LIN {X 0,Y 511.313,Z 919.131,A -85,B 0,C 180,E1 -11823.667,E2 -11823.667} C_VEL
LIN {X 0,Y 515.033,Z 901.309,A -85,B 0,C 180,E1 -11825.28,E2 -11825.28} C_VEL
LIN {X 0,Y 519.279,Z 879.68,A -85,B 0,C 180,E1 -11826.956,E2 -11826.956} C_VEL
LIN {X 0,Y 522.584,Z 861.401,A -85,B 0,C 180,E1 -11828.171,E2 -11828.171} C_VEL
LIN {X 0,Y 526.187,Z 839.915,A -85,B 0,C 180,E1 -11829.397,E2 -11829.397} C_VEL
LIN {X 0,Y 529.318,Z 818.14,A -85,B 0,C 180,E1 -11830.423,E2 -11830.423} C_VEL
LIN {X 0,Y 532.01,Z 796.933,A -85,B 0,C 180,E1 -11831.255,E2 -11831.255} C_VEL
LIN {X 0,Y 534.495,Z 772.49,A -85,B 0,C 180,E1 -11832.005,E2 -11832.005} C_VEL
LIN {X 0,Y 536.169,Z 751.43,A -85,B 0,C 180,E1 -11832.497,E2 -11832.497} C_VEL
LIN {X 0,Y 537.704,Z 719.028,A -85,B 0,C 180,E1 -11833.031,E2 -11833.031} C_VEL
LIN {X 0,Y 546.817,Z 464.332,A -85,B 0,C 180,E1 -11836.745,E2 -11836.745} C_VEL
LIN {X 0,Y 547.523,Z 441.329,A -85,B 0,C 180,E1 -11837.1,E2 -11837.1} C_VEL
LIN {X 0,Y 534.412,Z 419.937,A -85,B 0,C 180,E1 -11839.073,E2 -11839.073} C_VEL
LIN {X 0,Y 522.198,Z 402.674,A -85,B 0,C 180,E1 -11841.023,E2 -11841.023} C_VEL
LIN {X 0,Y 514.394,Z 392.307,A -85,B 0,C 180,E1 -11842.349,E2 -11842.349} C_VEL
LIN {X 0,Y 507.087,Z 382.771,A -85,B 0,C 180,E1 -11843.663,E2 -11843.663} C_VEL
LIN {X 0,Y 502.805,Z 377.333,A -85,B 0,C 180,E1 -11844.467,E2 -11844.467} C_VEL
LIN {X 0,Y 499.561,Z 373.172,A -85,B 0,C 180,E1 -11845.097,E2 -11845.097} C_VEL
LIN {X 0,Y 498.35,Z 371.8,A -85,B 0,C 180,E1 -11845.332,E2 -11845.332} C_VEL
LIN {X 0,Y 495.465,Z 368.374,A -85,B 0,C 180,E1 -11845.908,E2 -11845.908} C_VEL
LIN {X 0,Y 494.414,Z 366.395,A -85,B 0,C 180,E1 -11846.14,E2 -11846.14} C_VEL
LIN {X 0,Y 491.49,Z 364.03,A -85,B 0,C 180,E1 -11846.716,E2 -11846.716} C_VEL
LIN {X 0,Y 490.096,Z 361.064,A -85,B 0,C 180,E1 -11847.046,E2 -11847.046} C_VEL
LIN {X 0,Y 489.943,Z 360.201,A -85,B 0,C 180,E1 -11847.121,E2 -11847.121} C_VEL
LIN {X 0,Y 489.937,Z 360.204,A -85,B 0,C 180,E1 -11850.672,E2 -11850.672} C_VEL
LIN {X 0,Y 489.975,Z 360.197,A -85,B 0,C 180,E1 -11854.106,E2 -11854.106} C_VEL
LIN {X 0,Y 489.965,Z 360.19,A -85,B 0,C 180,E1 -11857.586,E2 -11857.586} C_VEL
LIN {X 0,Y 489.933,Z 360.182,A -85,B 0,C 180,E1 -11861.065,E2 -11861.065} C_VEL
LIN {X 0,Y 489.943,Z 360.174,A -85,B 0,C 180,E1 -11864.615,E2 -11864.615} C_VEL
LIN {X 0,Y 489.979,Z 360.18,A -85,B 0,C 180,E1 -11867.986,E2 -11867.986} C_VEL
LIN {X 0,Y 489.937,Z 360.202,A -85,B 0,C 180,E1 -11871.432,E2 -11871.432} C_VEL
LIN {X 0,Y 489.932,Z 360.192,A -85,B 0,C 180,E1 -11875.083,E2 -11875.083} C_VEL
LIN {X 0,Y 489.976,Z 360.169,A -85,B 0,C 180,E1 -11878.48,E2 -11878.48} C_VEL
LIN {X 0,Y 489.95,Z 360.185,A -85,B 0,C 180,E1 -11881.871,E2 -11881.871} C_VEL
LIN {X 0,Y 489.931,Z 360.202,A -85,B 0,C 180,E1 -11885.387,E2 -11885.387} C_VEL
LIN {X 0,Y 489.963,Z 360.181,A -85,B 0,C 180,E1 -11888.804,E2 -11888.804} C_VEL
LIN {X 0,Y 489.967,Z 360.172,A -85,B 0,C 180,E1 -11892.253,E2 -11892.253} C_VEL
LIN {X 0,Y 489.93,Z 360.186,A -85,B 0,C 180,E1 -11895.628,E2 -11895.628} C_VEL
LIN {X 0,Y 489.946,Z 360.196,A -85,B 0,C 180,E1 -11899.182,E2 -11899.182} C_VEL
LIN {X 0,Y 490,Z 360.194,A -85,B 0,C 180,E1 -11902.686,E2 -11902.686} C_VEL
LIN {X 0,Y 489.945,Z 360.2,A -85,B 0,C 180,E1 -11906.156,E2 -11906.156} C_VEL
LIN {X 0,Y 489.937,Z 360.204,A -85,B 0,C 180,E1 -11909.611,E2 -11909.611} C_VEL
LIN {X 0,Y 489.959,Z 360.296,A -85,B 0,C 180,E1 -11911.399,E2 -11911.399} C_VEL
LIN {X 0,Y 491.112,Z 363.479,A -85,B 0,C 180,E1 -11912.117,E2 -11912.117} C_VEL
LIN {X 0,Y 492.216,Z 365.12,A -85,B 0,C 180,E1 -11912.57,E2 -11912.57} C_VEL
LIN {X 0,Y 494.473,Z 369.884,A -85,B 0,C 180,E1 -11913.629,E2 -11913.629} C_VEL
LIN {X 0,Y 497.873,Z 374.385,A -85,B 0,C 180,E1 -11914.322,E2 -11914.322} C_VEL
LIN {X 0,Y 506.25,Z 385.924,A -85,B 0,C 180,E1 -11915.951,E2 -11915.951} C_VEL
LIN {X 0,Y 515.686,Z 399.295,A -85,B 0,C 180,E1 -11917.663,E2 -11917.663} C_VEL
LIN {X 0,Y 526.361,Z 415.198,A -85,B 0,C 180,E1 -11919.469,E2 -11919.469} C_VEL
LIN {X 0,Y 538.606,Z 435.059,A -85,B 0,C 180,E1 -11921.409,E2 -11921.409} C_VEL
LIN {X 0,Y 547.534,Z 450.875,A -85,B 0,C 180,E1 -11922.751,E2 -11922.751} C_VEL
LIN {X 0,Y 538.539,Z 702.351,A -85,B 0,C 180,E1 -11926.422,E2 -11926.422} C_VEL
LIN {X 0,Y 536.196,Z 765.178,A -85,B 0,C 180,E1 -11927.36,E2 -11927.36} C_VEL
LIN {X 0,Y 534.217,Z 790.289,A -85,B 0,C 180,E1 -11927.896,E2 -11927.896} C_VEL
LIN {X 0,Y 532.012,Z 811.704,A -85,B 0,C 180,E1 -11928.504,E2 -11928.504} C_VEL
LIN {X 0,Y 528.819,Z 836.909,A -85,B 0,C 180,E1 -11929.426,E2 -11929.426} C_VEL
LIN {X 0,Y 525.791,Z 857.705,A -85,B 0,C 180,E1 -11930.371,E2 -11930.371} C_VEL
LIN {X 0,Y 521.793,Z 881.818,A -85,B 0,C 180,E1 -11931.69,E2 -11931.69} C_VEL
LIN {X 0,Y 518.363,Z 900.79,A -85,B 0,C 180,E1 -11932.927,E2 -11932.927} C_VEL
LIN {X 0,Y 514.303,Z 921.939,A -85,B 0,C 180,E1 -11934.526,E2 -11934.526} C_VEL
LIN {X 0,Y 510.427,Z 940.778,A -85,B 0,C 180,E1 -11936.197,E2 -11936.197} C_VEL
LIN {X 0,Y 506.569,Z 959.339,A -85,B 0,C 180,E1 -11938.077,E2 -11938.077} C_VEL
LIN {X 0,Y 502.777,Z 977.115,A -85,B 0,C 180,E1 -11940.186,E2 -11940.186} C_VEL
LIN {X 0,Y 499.343,Z 993.821,A -85,B 0,C 180,E1 -11942.448,E2 -11942.448} C_VEL
LIN {X 0,Y 496.299,Z 1008.916,A -85,B 0,C 180,E1 -11944.843,E2 -11944.843} C_VEL
LIN {X 0,Y 493.733,Z 1022.841,A -85,B 0,C 180,E1 -11947.37,E2 -11947.37} C_VEL
LIN {X 0,Y 491.7,Z 1034.931,A -85,B 0,C 180,E1 -11949.968,E2 -11949.968} C_VEL
LIN {X 0,Y 490.163,Z 1045.803,A -85,B 0,C 180,E1 -11952.673,E2 -11952.673} C_VEL
LIN {X 0,Y 489.084,Z 1054.892,A -85,B 0,C 180,E1 -11955.436,E2 -11955.436} C_VEL
LIN {X 0,Y 488.449,Z 1062.177,A -85,B 0,C 180,E1 -11958.099,E2 -11958.099} C_VEL
LIN {X 0,Y 488.077,Z 1068.149,A -85,B 0,C 180,E1 -11960.924,E2 -11960.924} C_VEL
LIN {X 0,Y 487.956,Z 1071.916,A -85,B 0,C 180,E1 -11963.292,E2 -11963.292} C_VEL
LIN {X 0,Y 487.923,Z 1074.916,A -85,B 0,C 180,E1 -11966.005,E2 -11966.005} C_VEL
LIN {X 0,Y 487.926,Z 1076.286,A -85,B 0,C 180,E1 -11968.708,E2 -11968.708} C_VEL
LIN {X 0,Y 487.932,Z 1076.332,A -85,B 0,C 180,E1 -11971.057,E2 -11971.057} C_VEL
LIN {X 0,Y 487.925,Z 1075.157,A -85,B 0,C 180,E1 -11973.642,E2 -11973.642} C_VEL
LIN {X 0,Y 487.952,Z 1072.239,A -85,B 0,C 180,E1 -11976.471,E2 -11976.471} C_VEL
LIN {X 0,Y 488.061,Z 1068.568,A -85,B 0,C 180,E1 -11978.839,E2 -11978.839} C_VEL
LIN {X 0,Y 488.368,Z 1063.239,A -85,B 0,C 180,E1 -11981.455,E2 -11981.455} C_VEL
LIN {X 0,Y 488.988,Z 1055.838,A -85,B 0,C 180,E1 -11984.246,E2 -11984.246} C_VEL
LIN {X 0,Y 489.879,Z 1047.867,A -85,B 0,C 180,E1 -11986.726,E2 -11986.726} C_VEL
LIN {X 0,Y 491.42,Z 1036.727,A -85,B 0,C 180,E1 -11989.617,E2 -11989.617} C_VEL
LIN {X 0,Y 493.107,Z 1026.321,A -85,B 0,C 180,E1 -11991.907,E2 -11991.907} C_VEL
LIN {X 0,Y 495.582,Z 1012.759,A -85,B 0,C 180,E1 -11994.502,E2 -11994.502} C_VEL
LIN {X 0,Y 498.352,Z 998.474,A -85,B 0,C 180,E1 -11996.836,E2 -11996.836} C_VEL
LIN {X 0,Y 501.637,Z 982.689,A -85,B 0,C 180,E1 -11999.101,E2 -11999.101} C_VEL
LIN {X 0,Y 505.249,Z 965.34,A -85,B 0,C 180,E1 -12001.231,E2 -12001.231} C_VEL
LIN {X 0,Y 509.17,Z 946.864,A -85,B 0,C 180,E1 -12003.22,E2 -12003.22} C_VEL
LIN {X 0,Y 513.17,Z 927.247,A -85,B 0,C 180,E1 -12005.017,E2 -12005.017} C_VEL
LIN {X 0,Y 517.179,Z 907.204,A -85,B 0,C 180,E1 -12006.615,E2 -12006.615} C_VEL
LIN {X 0,Y 520.987,Z 886.248,A -85,B 0,C 180,E1 -12008.03,E2 -12008.03} C_VEL
LIN {X 0,Y 524.287,Z 867.033,A -85,B 0,C 180,E1 -12009.143,E2 -12009.143} C_VEL
LIN {X 0,Y 527.961,Z 842.844,A -85,B 0,C 180,E1 -12010.317,E2 -12010.317} C_VEL
LIN {X 0,Y 530.724,Z 822.066,A -85,B 0,C 180,E1 -12011.139,E2 -12011.139} C_VEL
LIN {X 0,Y 533.484,Z 797.595,A -85,B 0,C 180,E1 -12011.913,E2 -12011.913} C_VEL
LIN {X 0,Y 535.471,Z 774.643,A -85,B 0,C 180,E1 -12012.452,E2 -12012.452} C_VEL
LIN {X 0,Y 536.913,Z 748.928,A -85,B 0,C 180,E1 -12012.896,E2 -12012.896} C_VEL
LIN {X 0,Y 545.727,Z 498.186,A -85,B 0,C 180,E1 -12016.55,E2 -12016.55} C_VEL
LIN {X 0,Y 547.401,Z 450.448,A -85,B 0,C 180,E1 -12017.259,E2 -12017.259} C_VEL
LIN {X 0,Y 535.227,Z 429.465,A -85,B 0,C 180,E1 -12019.096,E2 -12019.096} C_VEL
LIN {X 0,Y 523.091,Z 410.309,A -85,B 0,C 180,E1 -12021.049,E2 -12021.049} C_VEL
LIN {X 0,Y 511.933,Z 393.825,A -85,B 0,C 180,E1 -12022.982,E2 -12022.982} C_VEL
LIN {X 0,Y 503.577,Z 382.206,A -85,B 0,C 180,E1 -12024.529,E2 -12024.529} C_VEL
LIN {X 0,Y 496.871,Z 373.305,A -85,B 0,C 180,E1 -12025.843,E2 -12025.843} C_VEL
LIN {X 0,Y 494.047,Z 368.955,A -85,B 0,C 180,E1 -12026.495,E2 -12026.495} C_VEL
LIN {X 0,Y 492.345,Z 365.591,A -85,B 0,C 180,E1 -12027.302,E2 -12027.302} C_VEL
LIN {X 0,Y 490.139,Z 361.244,A -85,B 0,C 180,E1 -12028.38,E2 -12028.38} C_VEL
LIN {X 0,Y 489.946,Z 360.176,A -85,B 0,C 180,E1 -12028.64,E2 -12028.64} C_VEL
LIN {X 0,Y 489.935,Z 360.177,A -85,B 0,C 180,E1 -12032.137,E2 -12032.137} C_VEL
LIN {X 0,Y 489.961,Z 360.177,A -85,B 0,C 180,E1 -12035.655,E2 -12035.655} C_VEL
LIN {X 0,Y 489.96,Z 360.184,A -85,B 0,C 180,E1 -12038.95,E2 -12038.95} C_VEL
LIN {X 0,Y 489.935,Z 360.2,A -85,B 0,C 180,E1 -12042.419,E2 -12042.419} C_VEL
LIN {X 0,Y 489.954,Z 360.203,A -85,B 0,C 180,E1 -12045.945,E2 -12045.945} C_VEL
LIN {X 0,Y 489.983,Z 360.182,A -85,B 0,C 180,E1 -12049.417,E2 -12049.417} C_VEL
LIN {X 0,Y 489.935,Z 360.172,A -85,B 0,C 180,E1 -12052.849,E2 -12052.849} C_VEL
LIN {X 0,Y 489.939,Z 360.185,A -85,B 0,C 180,E1 -12056.373,E2 -12056.373} C_VEL
LIN {X 0,Y 489.986,Z 360.198,A -85,B 0,C 180,E1 -12059.883,E2 -12059.883} C_VEL
LIN {X 0,Y 489.964,Z 360.186,A -85,B 0,C 180,E1 -12063.393,E2 -12063.393} C_VEL
LIN {X 0,Y 489.931,Z 360.174,A -85,B 0,C 180,E1 -12066.798,E2 -12066.798} C_VEL
LIN {X 0,Y 489.965,Z 360.183,A -85,B 0,C 180,E1 -12070.227,E2 -12070.227} C_VEL
LIN {X 0,Y 489.99,Z 360.198,A -85,B 0,C 180,E1 -12073.813,E2 -12073.813} C_VEL
LIN {X 0,Y 489.941,Z 360.194,A -85,B 0,C 180,E1 -12077.233,E2 -12077.233} C_VEL
LIN {X 0,Y 489.943,Z 360.182,A -85,B 0,C 180,E1 -12080.821,E2 -12080.821} C_VEL
LIN {X 0,Y 489.986,Z 360.174,A -85,B 0,C 180,E1 -12084.216,E2 -12084.216} C_VEL
LIN {X 0,Y 489.96,Z 360.178,A -85,B 0,C 180,E1 -12087.729,E2 -12087.729} C_VEL
LIN {X 0,Y 489.937,Z 360.181,A -85,B 0,C 180,E1 -12091.224,E2 -12091.224} C_VEL
LIN {X 0,Y 489.96,Z 360.317,A -85,B 0,C 180,E1 -12093.034,E2 -12093.034} C_VEL
LIN {X 0,Y 490.954,Z 363.217,A -85,B 0,C 180,E1 -12093.29,E2 -12093.29} C_VEL
LIN {X 0,Y 493.433,Z 365.836,A -85,B 0,C 180,E1 -12093.797,E2 -12093.797} C_VEL
LIN {X 0,Y 494.715,Z 366.871,A -85,B 0,C 180,E1 -12094.046,E2 -12094.046} C_VEL
LIN {X 0,Y 497.133,Z 370.66,A -85,B 0,C 180,E1 -12094.555,E2 -12094.555} C_VEL
LIN {X 0,Y 499.453,Z 372.962,A -85,B 0,C 180,E1 -12094.999,E2 -12094.999} C_VEL
LIN {X 0,Y 502.626,Z 377.161,A -85,B 0,C 180,E1 -12095.618,E2 -12095.618} C_VEL
LIN {X 0,Y 504.307,Z 379.254,A -85,B 0,C 180,E1 -12095.936,E2 -12095.936} C_VEL
LIN {X 0,Y 509.417,Z 385.807,A -85,B 0,C 180,E1 -12096.879,E2 -12096.879} C_VEL
LIN {X 0,Y 519.764,Z 399.344,A -85,B 0,C 180,E1 -12098.681,E2 -12098.681} C_VEL
LIN {X 0,Y 532.978,Z 417.831,A -85,B 0,C 180,E1 -12100.811,E2 -12100.811} C_VEL
LIN {X 0,Y 544.745,Z 436.73,A -85,B 0,C 180,E1 -12102.598,E2 -12102.598} C_VEL
LIN {X 0,Y 547.588,Z 441.89,A -85,B 0,C 180,E1 -12103.021,E2 -12103.021} C_VEL
LIN {X 0,Y 538.598,Z 691.495,A -85,B 0,C 180,E1 -12106.663,E2 -12106.663} C_VEL
LIN {X 0,Y 536.531,Z 745.384,A -85,B 0,C 180,E1 -12107.475,E2 -12107.475} C_VEL
LIN {X 0,Y 534.688,Z 769.631,A -85,B 0,C 180,E1 -12108.014,E2 -12108.014} C_VEL
LIN {X 0,Y 532.499,Z 791.967,A -85,B 0,C 180,E1 -12108.669,E2 -12108.669} C_VEL
LIN {X 0,Y 529.612,Z 815.624,A -85,B 0,C 180,E1 -12109.563,E2 -12109.563} C_VEL
LIN {X 0,Y 526.696,Z 836.1,A -85,B 0,C 180,E1 -12110.508,E2 -12110.508} C_VEL
LIN {X 0,Y 522.882,Z 859.553,A -85,B 0,C 180,E1 -12111.808,E2 -12111.808} C_VEL
LIN {X 0,Y 519.541,Z 878.086,A -85,B 0,C 180,E1 -12113.028,E2 -12113.028} C_VEL
LIN {X 0,Y 515.648,Z 898.366,A -85,B 0,C 180,E1 -12114.564,E2 -12114.564} C_VEL
LIN {X 0,Y 511.606,Z 917.639,A -85,B 0,C 180,E1 -12116.286,E2 -12116.286} C_VEL
LIN {X 0,Y 507.757,Z 935.822,A -85,B 0,C 180,E1 -12118.146,E2 -12118.146} C_VEL
LIN {X 0,Y 506.748,Z 940.366,A -85,B 0,C 180,E1 -12118.669,E2 -12118.669} C_VEL
LIN {X 0,Y 504.678,Z 945.91,A -85,B 0,C 180,E1 -12119.252,E2 -12119.252} C_VEL
LIN {X 0,Y 495.934,Z 960.386,A -85,B 0,C 180,E1 -12120.722,E2 -12120.722} C_VEL
LIN {X 0,Y 494.284,Z 964.589,A -85,B 0,C 180,E1 -12121.277,E2 -12121.277} C_VEL
LIN {X 0,Y 490.862,Z 979.995,A -85,B 0,C 180,E1 -12123.636,E2 -12123.636} C_VEL
LIN {X 0,Y 487.931,Z 993.479,A -85,B 0,C 180,E1 -12126.062,E2 -12126.062} C_VEL
LIN {X 0,Y 485.559,Z 1005.29,A -85,B 0,C 180,E1 -12128.497,E2 -12128.497} C_VEL
LIN {X 0,Y 483.479,Z 1016.797,A -85,B 0,C 180,E1 -12131.303,E2 -12131.303} C_VEL
LIN {X 0,Y 482.143,Z 1025.397,A -85,B 0,C 180,E1 -12133.78,E2 -12133.78} C_VEL
LIN {X 0,Y 481.037,Z 1033.999,A -85,B 0,C 180,E1 -12136.783,E2 -12136.783} C_VEL
LIN {X 0,Y 480.461,Z 1039.803,A -85,B 0,C 180,E1 -12139.326,E2 -12139.326} C_VEL
LIN {X 0,Y 480.12,Z 1044.781,A -85,B 0,C 180,E1 -12142.1,E2 -12142.1} C_VEL
LIN {X 0,Y 479.983,Z 1048.099,A -85,B 0,C 180,E1 -12144.861,E2 -12144.861} C_VEL
LIN {X 0,Y 479.937,Z 1049.885,A -85,B 0,C 180,E1 -12147.254,E2 -12147.254} C_VEL
LIN {X 0,Y 479.942,Z 1050.696,A -85,B 0,C 180,E1 -12150,E2 -12150} C_VEL
LIN {X 0,Y 479.939,Z 1049.937,A -85,B 0,C 180,E1 -12152.747,E2 -12152.747} C_VEL
LIN {X 0,Y 479.983,Z 1048.185,A -85,B 0,C 180,E1 -12155.139,E2 -12155.139} C_VEL
LIN {X 0,Y 480.112,Z 1044.91,A -85,B 0,C 180,E1 -12157.901,E2 -12157.901} C_VEL
LIN {X 0,Y 480.449,Z 1039.993,A -85,B 0,C 180,E1 -12160.674,E2 -12160.674} C_VEL
LIN {X 0,Y 481.016,Z 1034.226,A -85,B 0,C 180,E1 -12163.218,E2 -12163.218} C_VEL
LIN {X 0,Y 482.124,Z 1025.575,A -85,B 0,C 180,E1 -12166.259,E2 -12166.259} C_VEL
LIN {X 0,Y 483.428,Z 1017.131,A -85,B 0,C 180,E1 -12168.699,E2 -12168.699} C_VEL
LIN {X 0,Y 485.4,Z 1006.222,A -85,B 0,C 180,E1 -12171.394,E2 -12171.394} C_VEL
LIN {X 0,Y 487.841,Z 993.938,A -85,B 0,C 180,E1 -12173.943,E2 -12173.943} C_VEL
LIN {X 0,Y 490.757,Z 980.528,A -85,B 0,C 180,E1 -12176.37,E2 -12176.37} C_VEL
LIN {X 0,Y 494.052,Z 965.666,A -85,B 0,C 180,E1 -12178.663,E2 -12178.663} C_VEL
LIN {X 0,Y 497.486,Z 950.661,A -85,B 0,C 180,E1 -12180.698,E2 -12180.698} C_VEL
LIN {X 0,Y 501.626,Z 932.427,A -85,B 0,C 180,E1 -12182.832,E2 -12182.832} C_VEL
LIN {X 0,Y 505.356,Z 915.703,A -85,B 0,C 180,E1 -12184.532,E2 -12184.532} C_VEL
LIN {X 0,Y 509.862,Z 894.54,A -85,B 0,C 180,E1 -12186.387,E2 -12186.387} C_VEL
LIN {X 0,Y 513.524,Z 876.174,A -85,B 0,C 180,E1 -12187.765,E2 -12187.765} C_VEL
LIN {X 0,Y 517.549,Z 854.252,A -85,B 0,C 180,E1 -12189.18,E2 -12189.18} C_VEL
LIN {X 0,Y 520.985,Z 833.372,A -85,B 0,C 180,E1 -12190.299,E2 -12190.299} C_VEL
LIN {X 0,Y 524.289,Z 810.681,A -85,B 0,C 180,E1 -12191.326,E2 -12191.326} C_VEL
LIN {X 0,Y 527.081,Z 787.101,A -85,B 0,C 180,E1 -12192.166,E2 -12192.166} C_VEL
LIN {X 0,Y 529.455,Z 763.06,A -85,B 0,C 180,E1 -12192.838,E2 -12192.838} C_VEL
LIN {X 0,Y 531.053,Z 738.722,A -85,B 0,C 180,E1 -12193.319,E2 -12193.319} C_VEL
LIN {X 0,Y 540.023,Z 498.912,A -85,B 0,C 180,E1 -12196.856,E2 -12196.856} C_VEL
LIN {X 0,Y 541.977,Z 444.822,A -85,B 0,C 180,E1 -12197.671,E2 -12197.671} C_VEL
LIN {X 0,Y 529.659,Z 424.76,A -85,B 0,C 180,E1 -12199.574,E2 -12199.574} C_VEL
LIN {X 0,Y 518.068,Z 408.348,A -85,B 0,C 180,E1 -12201.47,E2 -12201.47} C_VEL
LIN {X 0,Y 507.851,Z 394.552,A -85,B 0,C 180,E1 -12203.27,E2 -12203.27} C_VEL
LIN {X 0,Y 499.417,Z 383.838,A -85,B 0,C 180,E1 -12204.858,E2 -12204.858} C_VEL
LIN {X 0,Y 495.264,Z 378.612,A -85,B 0,C 180,E1 -12205.682,E2 -12205.682} C_VEL
LIN {X 0,Y 492.058,Z 374.575,A -85,B 0,C 180,E1 -12206.341,E2 -12206.341} C_VEL
LIN {X 0,Y 490.964,Z 373.168,A -85,B 0,C 180,E1 -12206.571,E2 -12206.571} C_VEL
LIN {X 0,Y 488.016,Z 370.089,A -85,B 0,C 180,E1 -12207.185,E2 -12207.185} C_VEL
LIN {X 0,Y 486.42,Z 367.363,A -85,B 0,C 180,E1 -12207.553,E2 -12207.553} C_VEL
LIN {X 0,Y 483.499,Z 364.901,A -85,B 0,C 180,E1 -12208.173,E2 -12208.173} C_VEL
LIN {X 0,Y 482.144,Z 361.991,A -85,B 0,C 180,E1 -12208.517,E2 -12208.517} C_VEL
LIN {X 0,Y 481.997,Z 361.172,A -85,B 0,C 180,E1 -12208.58,E2 -12208.58} C_VEL
LIN {X 0,Y 482.04,Z 361.165,A -85,B 0,C 180,E1 -12212.044,E2 -12212.044} C_VEL
LIN {X 0,Y 482.028,Z 361.168,A -85,B 0,C 180,E1 -12215.619,E2 -12215.619} C_VEL
LIN {X 0,Y 481.994,Z 361.183,A -85,B 0,C 180,E1 -12218.99,E2 -12218.99} C_VEL
LIN {X 0,Y 482.015,Z 361.189,A -85,B 0,C 180,E1 -12222.495,E2 -12222.495} C_VEL
LIN {X 0,Y 482.057,Z 361.173,A -85,B 0,C 180,E1 -12226.077,E2 -12226.077} C_VEL
LIN {X 0,Y 482.015,Z 361.163,A -85,B 0,C 180,E1 -12229.723,E2 -12229.723} C_VEL
LIN {X 0,Y 481.991,Z 361.166,A -85,B 0,C 180,E1 -12233.209,E2 -12233.209} C_VEL
LIN {X 0,Y 482.01,Z 361.185,A -85,B 0,C 180,E1 -12236.789,E2 -12236.789} C_VEL
LIN {X 0,Y 482.058,Z 361.181,A -85,B 0,C 180,E1 -12240.357,E2 -12240.357} C_VEL
LIN {X 0,Y 482.011,Z 361.164,A -85,B 0,C 180,E1 -12243.925,E2 -12243.925} C_VEL
LIN {X 0,Y 481.989,Z 361.165,A -85,B 0,C 180,E1 -12247.424,E2 -12247.424} C_VEL
LIN {X 0,Y 482.02,Z 361.18,A -85,B 0,C 180,E1 -12250.881,E2 -12250.881} C_VEL
LIN {X 0,Y 482.047,Z 361.186,A -85,B 0,C 180,E1 -12254.413,E2 -12254.413} C_VEL
LIN {X 0,Y 481.996,Z 361.178,A -85,B 0,C 180,E1 -12257.88,E2 -12257.88} C_VEL
LIN {X 0,Y 481.992,Z 361.172,A -85,B 0,C 180,E1 -12261.542,E2 -12261.542} C_VEL
LIN {X 0,Y 482.032,Z 361.165,A -85,B 0,C 180,E1 -12264.977,E2 -12264.977} C_VEL
LIN {X 0,Y 482.029,Z 361.168,A -85,B 0,C 180,E1 -12268.496,E2 -12268.496} C_VEL
LIN {X 0,Y 482.029,Z 361.408,A -85,B 0,C 180,E1 -12270.078,E2 -12270.078} C_VEL
LIN {X 0,Y 483.601,Z 365.007,A -85,B 0,C 180,E1 -12270.986,E2 -12270.986} C_VEL
LIN {X 0,Y 484.337,Z 366.365,A -85,B 0,C 180,E1 -12271.349,E2 -12271.349} C_VEL
LIN {X 0,Y 485.86,Z 369.527,A -85,B 0,C 180,E1 -12272.07,E2 -12272.07} C_VEL
LIN {X 0,Y 491.716,Z 377.195,A -85,B 0,C 180,E1 -12273.336,E2 -12273.336} C_VEL
LIN {X 0,Y 502.133,Z 391.228,A -85,B 0,C 180,E1 -12275.431,E2 -12275.431} C_VEL
LIN {X 0,Y 512.492,Z 406.204,A -85,B 0,C 180,E1 -12277.357,E2 -12277.357} C_VEL
LIN {X 0,Y 522.524,Z 421.31,A -85,B 0,C 180,E1 -12279.089,E2 -12279.089} C_VEL
LIN {X 0,Y 534.415,Z 440.786,A -85,B 0,C 180,E1 -12281.015,E2 -12281.015} C_VEL
LIN {X 0,Y 541.967,Z 454.301,A -85,B 0,C 180,E1 -12282.18,E2 -12282.18} C_VEL
LIN {X 0,Y 532.673,Z 704.278,A -85,B 0,C 180,E1 -12285.858,E2 -12285.858} C_VEL
LIN {X 0,Y 530.305,Z 765.197,A -85,B 0,C 180,E1 -12286.776,E2 -12286.776} C_VEL
LIN {X 0,Y 528.266,Z 790.217,A -85,B 0,C 180,E1 -12287.315,E2 -12287.315} C_VEL
LIN {X 0,Y 526.015,Z 811.39,A -85,B 0,C 180,E1 -12287.919,E2 -12287.919} C_VEL
LIN {X 0,Y 522.7,Z 836.7,A -85,B 0,C 180,E1 -12288.849,E2 -12288.849} C_VEL
LIN {X 0,Y 519.602,Z 857.259,A -85,B 0,C 180,E1 -12289.788,E2 -12289.788} C_VEL
LIN {X 0,Y 515.582,Z 880.7,A -85,B 0,C 180,E1 -12291.072,E2 -12291.072} C_VEL
LIN {X 0,Y 511.845,Z 900.604,A -85,B 0,C 180,E1 -12292.377,E2 -12292.377} C_VEL
LIN {X 0,Y 507.67,Z 921.53,A -85,B 0,C 180,E1 -12293.971,E2 -12293.971} C_VEL
LIN {X 0,Y 503.598,Z 940.562,A -85,B 0,C 180,E1 -12295.675,E2 -12295.675} C_VEL
LIN {X 0,Y 499.6,Z 959.004,A -85,B 0,C 180,E1 -12297.563,E2 -12297.563} C_VEL
LIN {X 0,Y 495.596,Z 976.896,A -85,B 0,C 180,E1 -12299.709,E2 -12299.709} C_VEL
LIN {X 0,Y 492.004,Z 993.601,A -85,B 0,C 180,E1 -12302.001,E2 -12302.001} C_VEL
LIN {X 0,Y 488.8,Z 1008.697,A -85,B 0,C 180,E1 -12304.429,E2 -12304.429} C_VEL
LIN {X 0,Y 486.102,Z 1022.622,A -85,B 0,C 180,E1 -12306.994,E2 -12306.994} C_VEL
LIN {X 0,Y 483.996,Z 1034.424,A -85,B 0,C 180,E1 -12309.565,E2 -12309.565} C_VEL
LIN {X 0,Y 482.424,Z 1044.656,A -85,B 0,C 180,E1 -12312.136,E2 -12312.136} C_VEL
LIN {X 0,Y 481.242,Z 1053.956,A -85,B 0,C 180,E1 -12314.947,E2 -12314.947} C_VEL
LIN {X 0,Y 480.58,Z 1060.646,A -85,B 0,C 180,E1 -12317.381,E2 -12317.381} C_VEL
LIN {X 0,Y 480.148,Z 1067.091,A -85,B 0,C 180,E1 -12320.289,E2 -12320.289} C_VEL
LIN {X 0,Y 479.982,Z 1071.376,A -85,B 0,C 180,E1 -12322.94,E2 -12322.94} C_VEL
LIN {X 0,Y 479.934,Z 1074.124,A -85,B 0,C 180,E1 -12325.339,E2 -12325.339} C_VEL
LIN {X 0,Y 479.923,Z 1075.978,A -85,B 0,C 180,E1 -12328.209,E2 -12328.209} C_VEL
LIN {X 0,Y 479.93,Z 1076.165,A -85,B 0,C 180,E1 -12330.836,E2 -12330.836} C_VEL
LIN {X 0,Y 479.935,Z 1075.222,A -85,B 0,C 180,E1 -12333.225,E2 -12333.225} C_VEL
LIN {X 0,Y 479.952,Z 1072.675,A -85,B 0,C 180,E1 -12336.099,E2 -12336.099} C_VEL
LIN {X 0,Y 480.057,Z 1068.773,A -85,B 0,C 180,E1 -12338.746,E2 -12338.746} C_VEL
LIN {X 0,Y 480.343,Z 1063.799,A -85,B 0,C 180,E1 -12341.284,E2 -12341.284} C_VEL
LIN {X 0,Y 481.014,Z 1056.103,A -85,B 0,C 180,E1 -12344.322,E2 -12344.322} C_VEL
LIN {X 0,Y 481.957,Z 1048.058,A -85,B 0,C 180,E1 -12346.885,E2 -12346.885} C_VEL
LIN {X 0,Y 483.488,Z 1037.549,A -85,B 0,C 180,E1 -12349.7,E2 -12349.7} C_VEL
LIN {X 0,Y 485.326,Z 1026.68,A -85,B 0,C 180,E1 -12352.149,E2 -12352.149} C_VEL
LIN {X 0,Y 487.925,Z 1013.194,A -85,B 0,C 180,E1 -12354.792,E2 -12354.792} C_VEL
LIN {X 0,Y 490.796,Z 999.03,A -85,B 0,C 180,E1 -12357.152,E2 -12357.152} C_VEL
LIN {X 0,Y 494.211,Z 983.335,A -85,B 0,C 180,E1 -12359.448,E2 -12359.448} C_VEL
LIN {X 0,Y 497.964,Z 966.139,A -85,B 0,C 180,E1 -12361.606,E2 -12361.606} C_VEL
LIN {X 0,Y 501.646,Z 949.438,A -85,B 0,C 180,E1 -12363.444,E2 -12363.444} C_VEL
LIN {X 0,Y 506.031,Z 929.042,A -85,B 0,C 180,E1 -12365.377,E2 -12365.377} C_VEL
LIN {X 0,Y 509.72,Z 911.235,A -85,B 0,C 180,E1 -12366.836,E2 -12366.836} C_VEL
LIN {X 0,Y 514.093,Z 888.742,A -85,B 0,C 180,E1 -12368.419,E2 -12368.419} C_VEL
LIN {X 0,Y 517.549,Z 869.399,A -85,B 0,C 180,E1 -12369.569,E2 -12369.569} C_VEL
LIN {X 0,Y 521.233,Z 846.85,A -85,B 0,C 180,E1 -12370.71,E2 -12370.71} C_VEL
LIN {X 0,Y 524.399,Z 823.908,A -85,B 0,C 180,E1 -12371.644,E2 -12371.644} C_VEL
LIN {X 0,Y 527.109,Z 801.479,A -85,B 0,C 180,E1 -12372.381,E2 -12372.381} C_VEL
LIN {X 0,Y 529.396,Z 776.693,A -85,B 0,C 180,E1 -12372.992,E2 -12372.992} C_VEL
LIN {X 0,Y 530.834,Z 753.767,A -85,B 0,C 180,E1 -12373.406,E2 -12373.406} C_VEL
LIN {X 0,Y 540.011,Z 503.624,A -85,B 0,C 180,E1 -12377.085,E2 -12377.085} C_VEL
LIN {X 0,Y 541.805,Z 453.875,A -85,B 0,C 180,E1 -12377.833,E2 -12377.833} C_VEL
LIN {X 0,Y 530.241,Z 433.847,A -85,B 0,C 180,E1 -12379.628,E2 -12379.628} C_VEL
LIN {X 0,Y 517.391,Z 413.388,A -85,B 0,C 180,E1 -12381.764,E2 -12381.764} C_VEL
LIN {X 0,Y 505.056,Z 395.347,A -85,B 0,C 180,E1 -12383.985,E2 -12383.985} C_VEL
LIN {X 0,Y 494.553,Z 380.87,A -85,B 0,C 180,E1 -12386.046,E2 -12386.046} C_VEL
LIN {X 0,Y 489.87,Z 374.81,A -85,B 0,C 180,E1 -12387.02,E2 -12387.02} C_VEL
LIN {X 0,Y 485.406,Z 368.945,A -85,B 0,C 180,E1 -12388,E2 -12388} C_VEL
LIN {X 0,Y 483.813,Z 365.281,A -85,B 0,C 180,E1 -12388.891,E2 -12388.891} C_VEL
LIN {X 0,Y 482.174,Z 362.076,A -85,B 0,C 180,E1 -12389.741,E2 -12389.741} C_VEL
LIN {X 0,Y 481.997,Z 361.176,A -85,B 0,C 180,E1 -12390.003,E2 -12390.003} C_VEL
LIN {X 0,Y 482.043,Z 361.17,A -85,B 0,C 180,E1 -12393.382,E2 -12393.382} C_VEL
LIN {X 0,Y 482.023,Z 361.173,A -85,B 0,C 180,E1 -12396.917,E2 -12396.917} C_VEL
LIN {X 0,Y 481.992,Z 361.171,A -85,B 0,C 180,E1 -12400.362,E2 -12400.362} C_VEL
LIN {X 0,Y 482.016,Z 361.164,A -85,B 0,C 180,E1 -12403.861,E2 -12403.861} C_VEL
LIN {X 0,Y 482.04,Z 361.167,A -85,B 0,C 180,E1 -12407.298,E2 -12407.298} C_VEL
LIN {X 0,Y 482.001,Z 361.19,A -85,B 0,C 180,E1 -12410.809,E2 -12410.809} C_VEL
LIN {X 0,Y 481.999,Z 361.184,A -85,B 0,C 180,E1 -12414.405,E2 -12414.405} C_VEL
LIN {X 0,Y 482.036,Z 361.159,A -85,B 0,C 180,E1 -12417.86,E2 -12417.86} C_VEL
LIN {X 0,Y 482.01,Z 361.169,A -85,B 0,C 180,E1 -12421.189,E2 -12421.189} C_VEL
LIN {X 0,Y 481.997,Z 361.19,A -85,B 0,C 180,E1 -12424.76,E2 -12424.76} C_VEL
LIN {X 0,Y 482.024,Z 361.175,A -85,B 0,C 180,E1 -12428.229,E2 -12428.229} C_VEL
LIN {X 0,Y 482.04,Z 361.158,A -85,B 0,C 180,E1 -12431.746,E2 -12431.746} C_VEL
LIN {X 0,Y 481.999,Z 361.169,A -85,B 0,C 180,E1 -12435.152,E2 -12435.152} C_VEL
LIN {X 0,Y 482.005,Z 361.183,A -85,B 0,C 180,E1 -12438.756,E2 -12438.756} C_VEL
LIN {X 0,Y 482.059,Z 361.186,A -85,B 0,C 180,E1 -12442.179,E2 -12442.179} C_VEL
LIN {X 0,Y 482.034,Z 361.186,A -85,B 0,C 180,E1 -12445.824,E2 -12445.824} C_VEL
LIN {X 0,Y 482.004,Z 361.187,A -85,B 0,C 180,E1 -12449.312,E2 -12449.312} C_VEL
LIN {X 0,Y 482.023,Z 361.292,A -85,B 0,C 180,E1 -12451.569,E2 -12451.569} C_VEL
LIN {X 0,Y 483.085,Z 364.262,A -85,B 0,C 180,E1 -12451.857,E2 -12451.857} C_VEL
LIN {X 0,Y 485.739,Z 366.965,A -85,B 0,C 180,E1 -12452.435,E2 -12452.435} C_VEL
LIN {X 0,Y 486.88,Z 367.958,A -85,B 0,C 180,E1 -12452.674,E2 -12452.674} C_VEL
LIN {X 0,Y 489.267,Z 371.683,A -85,B 0,C 180,E1 -12453.209,E2 -12453.209} C_VEL
LIN {X 0,Y 491.764,Z 374.063,A -85,B 0,C 180,E1 -12453.717,E2 -12453.717} C_VEL
LIN {X 0,Y 494.822,Z 378.197,A -85,B 0,C 180,E1 -12454.353,E2 -12454.353} C_VEL
LIN {X 0,Y 496.593,Z 380.201,A -85,B 0,C 180,E1 -12454.703,E2 -12454.703} C_VEL
LIN {X 0,Y 501.667,Z 386.773,A -85,B 0,C 180,E1 -12455.697,E2 -12455.697} C_VEL
LIN {X 0,Y 508.743,Z 395.724,A -85,B 0,C 180,E1 -12457.007,E2 -12457.007} C_VEL
LIN {X 0,Y 521.083,Z 412.531,A -85,B 0,C 180,E1 -12459.147,E2 -12459.147} C_VEL
LIN {X 0,Y 532.135,Z 428.663,A -85,B 0,C 180,E1 -12460.925,E2 -12460.925} C_VEL
LIN {X 0,Y 542.037,Z 445.304,A -85,B 0,C 180,E1 -12462.449,E2 -12462.449} C_VEL
LIN {X 0,Y 532.672,Z 695.5,A -85,B 0,C 180,E1 -12466.128,E2 -12466.128} C_VEL
LIN {X 0,Y 530.636,Z 746.15,A -85,B 0,C 180,E1 -12466.9,E2 -12466.9} C_VEL
LIN {X 0,Y 528.71,Z 770.379,A -85,B 0,C 180,E1 -12467.447,E2 -12467.447} C_VEL
LIN {X 0,Y 526.374,Z 793.425,A -85,B 0,C 180,E1 -12468.132,E2 -12468.132} C_VEL
LIN {X 0,Y 523.411,Z 816.551,A -85,B 0,C 180,E1 -12469.022,E2 -12469.022} C_VEL
LIN {X 0,Y 520.493,Z 836.323,A -85,B 0,C 180,E1 -12469.943,E2 -12469.943} C_VEL
LIN {X 0,Y 516.581,Z 859.564,A -85,B 0,C 180,E1 -12471.24,E2 -12471.24} C_VEL
LIN {X 0,Y 513.079,Z 878.305,A -85,B 0,C 180,E1 -12472.482,E2 -12472.482} C_VEL
LIN {X 0,Y 509.037,Z 898.589,A -85,B 0,C 180,E1 -12474.033,E2 -12474.033} C_VEL
LIN {X 0,Y 504.837,Z 917.862,A -85,B 0,C 180,E1 -12475.772,E2 -12475.772} C_VEL
LIN {X 0,Y 500.817,Z 936.045,A -85,B 0,C 180,E1 -12477.652,E2 -12477.652} C_VEL
LIN {X 0,Y 496.984,Z 952.753,A -85,B 0,C 180,E1 -12479.669,E2 -12479.669} C_VEL
LIN {X 0,Y 494.284,Z 964.589,A -85,B 0,C 180,E1 -12481.277,E2 -12481.277} C_VEL
LIN {X 0,Y 492.271,Z 969.611,A -85,B 0,C 180,E1 -12481.937,E2 -12481.937} C_VEL
LIN {X 0,Y 483.654,Z 982.488,A -85,B 0,C 180,E1 -12483.64,E2 -12483.64} C_VEL
LIN {X 0,Y 482.108,Z 986.206,A -85,B 0,C 180,E1 -12484.261,E2 -12484.261} C_VEL
LIN {X 0,Y 479.111,Z 999.856,A -85,B 0,C 180,E1 -12486.899,E2 -12486.899} C_VEL
LIN {X 0,Y 476.792,Z 1011.242,A -85,B 0,C 180,E1 -12489.499,E2 -12489.499} C_VEL
LIN {X 0,Y 474.907,Z 1021.908,A -85,B 0,C 180,E1 -12492.351,E2 -12492.351} C_VEL
LIN {X 0,Y 473.625,Z 1030.263,A -85,B 0,C 180,E1 -12495.075,E2 -12495.075} C_VEL
LIN {X 0,Y 472.767,Z 1037.494,A -85,B 0,C 180,E1 -12497.914,E2 -12497.914} C_VEL
LIN {X 0,Y 472.266,Z 1042.974,A -85,B 0,C 180,E1 -12500.74,E2 -12500.74} C_VEL
LIN {X 0,Y 472.055,Z 1046.726,A -85,B 0,C 180,E1 -12503.31,E2 -12503.31} C_VEL
LIN {X 0,Y 471.96,Z 1049.632,A -85,B 0,C 180,E1 -12506.356,E2 -12506.356} C_VEL
LIN {X 0,Y 471.94,Z 1050.731,A -85,B 0,C 180,E1 -12509.029,E2 -12509.029} C_VEL
LIN {X 0,Y 471.936,Z 1050.638,A -85,B 0,C 180,E1 -12511.578,E2 -12511.578} C_VEL
LIN {X 0,Y 471.979,Z 1048.956,A -85,B 0,C 180,E1 -12514.618,E2 -12514.618} C_VEL
LIN {X 0,Y 472.086,Z 1046.219,A -85,B 0,C 180,E1 -12517.179,E2 -12517.179} C_VEL
LIN {X 0,Y 472.37,Z 1041.911,A -85,B 0,C 180,E1 -12519.996,E2 -12519.996} C_VEL
LIN {X 0,Y 472.964,Z 1035.633,A -85,B 0,C 180,E1 -12522.95,E2 -12522.95} C_VEL
LIN {X 0,Y 473.841,Z 1028.788,A -85,B 0,C 180,E1 -12525.545,E2 -12525.545} C_VEL
LIN {X 0,Y 475.357,Z 1019.156,A -85,B 0,C 180,E1 -12528.519,E2 -12528.519} C_VEL
LIN {X 0,Y 477.127,Z 1009.58,A -85,B 0,C 180,E1 -12530.999,E2 -12530.999} C_VEL
LIN {X 0,Y 479.799,Z 996.663,A -85,B 0,C 180,E1 -12533.847,E2 -12533.847} C_VEL
LIN {X 0,Y 482.609,Z 984.041,A -85,B 0,C 180,E1 -12536.219,E2 -12536.219} C_VEL
LIN {X 0,Y 486.275,Z 968.392,A -85,B 0,C 180,E1 -12538.761,E2 -12538.761} C_VEL
LIN {X 0,Y 489.78,Z 953.627,A -85,B 0,C 180,E1 -12540.825,E2 -12540.825} C_VEL
LIN {X 0,Y 493.911,Z 936.41,A -85,B 0,C 180,E1 -12542.937,E2 -12542.937} C_VEL
LIN {X 0,Y 498.005,Z 918.67,A -85,B 0,C 180,E1 -12544.796,E2 -12544.796} C_VEL
LIN {X 0,Y 502.133,Z 900.409,A -85,B 0,C 180,E1 -12546.47,E2 -12546.47} C_VEL
LIN {X 0,Y 506.431,Z 879.901,A -85,B 0,C 180,E1 -12548.075,E2 -12548.075} C_VEL
LIN {X 0,Y 509.942,Z 861.821,A -85,B 0,C 180,E1 -12549.297,E2 -12549.297} C_VEL
LIN {X 0,Y 513.809,Z 840.329,A -85,B 0,C 180,E1 -12550.54,E2 -12550.54} C_VEL
LIN {X 0,Y 517.061,Z 819.219,A -85,B 0,C 180,E1 -12551.551,E2 -12551.551} C_VEL
LIN {X 0,Y 519.831,Z 798.885,A -85,B 0,C 180,E1 -12552.365,E2 -12552.365} C_VEL
LIN {X 0,Y 522.627,Z 773.539,A -85,B 0,C 180,E1 -12553.164,E2 -12553.164} C_VEL
LIN {X 0,Y 524.433,Z 752.307,A -85,B 0,C 180,E1 -12553.669,E2 -12553.669} C_VEL
LIN {X 0,Y 526.004,Z 722.32,A -85,B 0,C 180,E1 -12554.178,E2 -12554.178} C_VEL
LIN {X 0,Y 535.832,Z 468.021,A -85,B 0,C 180,E1 -12557.943,E2 -12557.943} C_VEL
LIN {X 0,Y 536.52,Z 448.522,A -85,B 0,C 180,E1 -12558.245,E2 -12558.245} C_VEL
LIN {X 0,Y 525.3,Z 430.096,A -85,B 0,C 180,E1 -12560.027,E2 -12560.027} C_VEL
LIN {X 0,Y 511.827,Z 410.885,A -85,B 0,C 180,E1 -12562.304,E2 -12562.304} C_VEL
LIN {X 0,Y 500.51,Z 395.962,A -85,B 0,C 180,E1 -12564.384,E2 -12564.384} C_VEL
LIN {X 0,Y 495.675,Z 389.878,A -85,B 0,C 180,E1 -12565.329,E2 -12565.329} C_VEL
LIN {X 0,Y 492.074,Z 385.27,A -85,B 0,C 180,E1 -12566.062,E2 -12566.062} C_VEL
LIN {X 0,Y 487.813,Z 379.943,A -85,B 0,C 180,E1 -12566.959,E2 -12566.959} C_VEL
LIN {X 0,Y 484.579,Z 376.114,A -85,B 0,C 180,E1 -12567.66,E2 -12567.66} C_VEL
LIN {X 0,Y 483.309,Z 374.301,A -85,B 0,C 180,E1 -12567.95,E2 -12567.95} C_VEL
LIN {X 0,Y 480.239,Z 371.143,A -85,B 0,C 180,E1 -12568.633,E2 -12568.633} C_VEL
LIN {X 0,Y 478.717,Z 368.468,A -85,B 0,C 180,E1 -12569.012,E2 -12569.012} C_VEL
LIN {X 0,Y 475.79,Z 366.153,A -85,B 0,C 180,E1 -12569.675,E2 -12569.675} C_VEL
LIN {X 0,Y 474.294,Z 363.194,A -85,B 0,C 180,E1 -12570.076,E2 -12570.076} C_VEL
LIN {X 0,Y 474.087,Z 362.168,A -85,B 0,C 180,E1 -12570.179,E2 -12570.179} C_VEL
LIN {X 0,Y 474.099,Z 362.163,A -85,B 0,C 180,E1 -12573.681,E2 -12573.681} C_VEL
LIN {X 0,Y 474.06,Z 362.162,A -85,B 0,C 180,E1 -12577.179,E2 -12577.179} C_VEL
LIN {X 0,Y 474.057,Z 362.156,A -85,B 0,C 180,E1 -12580.897,E2 -12580.897} C_VEL
LIN {X 0,Y 474.09,Z 362.148,A -85,B 0,C 180,E1 -12584.338,E2 -12584.338} C_VEL
LIN {X 0,Y 474.089,Z 362.161,A -85,B 0,C 180,E1 -12587.824,E2 -12587.824} C_VEL
LIN {X 0,Y 474.058,Z 362.18,A -85,B 0,C 180,E1 -12591.387,E2 -12591.387} C_VEL
LIN {X 0,Y 474.056,Z 362.166,A -85,B 0,C 180,E1 -12595.039,E2 -12595.039} C_VEL
LIN {X 0,Y 474.091,Z 362.146,A -85,B 0,C 180,E1 -12598.55,E2 -12598.55} C_VEL
LIN {X 0,Y 474.076,Z 362.159,A -85,B 0,C 180,E1 -12601.934,E2 -12601.934} C_VEL
LIN {X 0,Y 474.055,Z 362.181,A -85,B 0,C 180,E1 -12605.446,E2 -12605.446} C_VEL
LIN {X 0,Y 474.07,Z 362.162,A -85,B 0,C 180,E1 -12608.979,E2 -12608.979} C_VEL
LIN {X 0,Y 474.106,Z 362.147,A -85,B 0,C 180,E1 -12612.546,E2 -12612.546} C_VEL
LIN {X 0,Y 474.062,Z 362.156,A -85,B 0,C 180,E1 -12615.914,E2 -12615.914} C_VEL
LIN {X 0,Y 474.056,Z 362.167,A -85,B 0,C 180,E1 -12619.469,E2 -12619.469} C_VEL
LIN {X 0,Y 474.094,Z 362.172,A -85,B 0,C 180,E1 -12622.966,E2 -12622.966} C_VEL
LIN {X 0,Y 474.1,Z 362.173,A -85,B 0,C 180,E1 -12626.59,E2 -12626.59} C_VEL
LIN {X 0,Y 474.108,Z 362.211,A -85,B 0,C 180,E1 -12628.603,E2 -12628.603} C_VEL
LIN {X 0,Y 475.374,Z 365.667,A -85,B 0,C 180,E1 -12629.485,E2 -12629.485} C_VEL
LIN {X 0,Y 476.42,Z 367.219,A -85,B 0,C 180,E1 -12629.967,E2 -12629.967} C_VEL
LIN {X 0,Y 477.295,Z 369.233,A -85,B 0,C 180,E1 -12630.393,E2 -12630.393} C_VEL
LIN {X 0,Y 484.762,Z 378.802,A -85,B 0,C 180,E1 -12632.117,E2 -12632.117} C_VEL
LIN {X 0,Y 489.03,Z 384.475,A -85,B 0,C 180,E1 -12633.049,E2 -12633.049} C_VEL
LIN {X 0,Y 496.157,Z 394.13,A -85,B 0,C 180,E1 -12634.527,E2 -12634.527} C_VEL
LIN {X 0,Y 507.009,Z 409.469,A -85,B 0,C 180,E1 -12636.618,E2 -12636.618} C_VEL
LIN {X 0,Y 518.913,Z 427.762,A -85,B 0,C 180,E1 -12638.738,E2 -12638.738} C_VEL
LIN {X 0,Y 530.84,Z 447.486,A -85,B 0,C 180,E1 -12640.708,E2 -12640.708} C_VEL
LIN {X 0,Y 536.452,Z 457.823,A -85,B 0,C 180,E1 -12641.6,E2 -12641.6} C_VEL
LIN {X 0,Y 526.839,Z 706.771,A -85,B 0,C 180,E1 -12645.289,E2 -12645.289} C_VEL
LIN {X 0,Y 524.471,Z 765.216,A -85,B 0,C 180,E1 -12646.179,E2 -12646.179} C_VEL
LIN {X 0,Y 522.37,Z 790.144,A -85,B 0,C 180,E1 -12646.72,E2 -12646.72} C_VEL
LIN {X 0,Y 520.074,Z 811.076,A -85,B 0,C 180,E1 -12647.321,E2 -12647.321} C_VEL
LIN {X 0,Y 516.84,Z 835.202,A -85,B 0,C 180,E1 -12648.204,E2 -12648.204} C_VEL
LIN {X 0,Y 513.805,Z 854.777,A -85,B 0,C 180,E1 -12649.092,E2 -12649.092} C_VEL
LIN {X 0,Y 509.994,Z 876.814,A -85,B 0,C 180,E1 -12650.271,E2 -12650.271} C_VEL
LIN {X 0,Y 505.88,Z 897.941,A -85,B 0,C 180,E1 -12651.638,E2 -12651.638} C_VEL
LIN {X 0,Y 501.898,Z 917.209,A -85,B 0,C 180,E1 -12653.083,E2 -12653.083} C_VEL
LIN {X 0,Y 497.334,Z 938.003,A -85,B 0,C 180,E1 -12654.913,E2 -12654.913} C_VEL
LIN {X 0,Y 493.52,Z 954.815,A -85,B 0,C 180,E1 -12656.621,E2 -12656.621} C_VEL
LIN {X 0,Y 489.121,Z 973.872,A -85,B 0,C 180,E1 -12658.855,E2 -12658.855} C_VEL
LIN {X 0,Y 485.615,Z 989.127,A -85,B 0,C 180,E1 -12660.927,E2 -12660.927} C_VEL
LIN {X 0,Y 482.117,Z 1004.933,A -85,B 0,C 180,E1 -12663.386,E2 -12663.386} C_VEL
LIN {X 0,Y 479.355,Z 1017.919,A -85,B 0,C 180,E1 -12665.737,E2 -12665.737} C_VEL
LIN {X 0,Y 476.933,Z 1030.535,A -85,B 0,C 180,E1 -12668.347,E2 -12668.347} C_VEL
LIN {X 0,Y 475.015,Z 1041.643,A -85,B 0,C 180,E1 -12671.085,E2 -12671.085} C_VEL
LIN {X 0,Y 473.713,Z 1050.729,A -85,B 0,C 180,E1 -12673.696,E2 -12673.696} C_VEL
LIN {X 0,Y 472.747,Z 1059.196,A -85,B 0,C 180,E1 -12676.671,E2 -12676.671} C_VEL
LIN {X 0,Y 472.268,Z 1065.076,A -85,B 0,C 180,E1 -12679.232,E2 -12679.232} C_VEL
LIN {X 0,Y 471.994,Z 1070.345,A -85,B 0,C 180,E1 -12682.208,E2 -12682.208} C_VEL
LIN {X 0,Y 471.943,Z 1073.447,A -85,B 0,C 180,E1 -12684.773,E2 -12684.773} C_VEL
LIN {X 0,Y 471.933,Z 1075.288,A -85,B 0,C 180,E1 -12687.207,E2 -12687.207} C_VEL
LIN {X 0,Y 471.944,Z 1076.105,A -85,B 0,C 180,E1 -12690,E2 -12690} C_VEL
LIN {X 0,Y 471.933,Z 1075.286,A -85,B 0,C 180,E1 -12692.793,E2 -12692.793} C_VEL
LIN {X 0,Y 471.942,Z 1073.408,A -85,B 0,C 180,E1 -12695.265,E2 -12695.265} C_VEL
LIN {X 0,Y 472.022,Z 1069.818,A -85,B 0,C 180,E1 -12698.159,E2 -12698.159} C_VEL
LIN {X 0,Y 472.301,Z 1064.618,A -85,B 0,C 180,E1 -12700.984,E2 -12700.984} C_VEL
LIN {X 0,Y 472.812,Z 1058.571,A -85,B 0,C 180,E1 -12703.576,E2 -12703.576} C_VEL
LIN {X 0,Y 473.814,Z 1049.895,A -85,B 0,C 180,E1 -12706.552,E2 -12706.552} C_VEL
LIN {X 0,Y 475.13,Z 1040.913,A -85,B 0,C 180,E1 -12709.108,E2 -12709.108} C_VEL
LIN {X 0,Y 477.242,Z 1028.782,A -85,B 0,C 180,E1 -12712.026,E2 -12712.026} C_VEL
LIN {X 0,Y 479.484,Z 1017.256,A -85,B 0,C 180,E1 -12714.387,E2 -12714.387} C_VEL
LIN {X 0,Y 482.603,Z 1002.703,A -85,B 0,C 180,E1 -12716.984,E2 -12716.984} C_VEL
LIN {X 0,Y 485.87,Z 987.92,A -85,B 0,C 180,E1 -12719.241,E2 -12719.241} C_VEL
LIN {X 0,Y 489.807,Z 971.019,A -85,B 0,C 180,E1 -12721.506,E2 -12721.506} C_VEL
LIN {X 0,Y 493.874,Z 953.134,A -85,B 0,C 180,E1 -12723.553,E2 -12723.553} C_VEL
LIN {X 0,Y 497.909,Z 935.368,A -85,B 0,C 180,E1 -12725.335,E2 -12725.335} C_VEL
LIN {X 0,Y 502.348,Z 914.894,A -85,B 0,C 180,E1 -12727.092,E2 -12727.092} C_VEL
LIN {X 0,Y 506.203,Z 896.202,A -85,B 0,C 180,E1 -12728.478,E2 -12728.478} C_VEL
LIN {X 0,Y 510.528,Z 873.542,A -85,B 0,C 180,E1 -12729.906,E2 -12729.906} C_VEL
LIN {X 0,Y 513.975,Z 853.489,A -85,B 0,C 180,E1 -12730.965,E2 -12730.965} C_VEL
LIN {X 0,Y 517.434,Z 831.103,A -85,B 0,C 180,E1 -12731.96,E2 -12731.96} C_VEL
LIN {X 0,Y 520.362,Z 808.209,A -85,B 0,C 180,E1 -12732.762,E2 -12732.762} C_VEL
LIN {X 0,Y 522.627,Z 787.224,A -85,B 0,C 180,E1 -12733.347,E2 -12733.347} C_VEL
LIN {X 0,Y 524.634,Z 761.045,A -85,B 0,C 180,E1 -12733.884,E2 -12733.884} C_VEL
LIN {X 0,Y 533.324,Z 534.551,A -85,B 0,C 180,E1 -12737.256,E2 -12737.256} C_VEL
LIN {X 0,Y 536.3,Z 457.275,A -85,B 0,C 180,E1 -12738.414,E2 -12738.414} C_VEL
LIN {X 0,Y 524.332,Z 436.592,A -85,B 0,C 180,E1 -12740.33,E2 -12740.33} C_VEL
LIN {X 0,Y 512.884,Z 418.448,A -85,B 0,C 180,E1 -12742.289,E2 -12742.289} C_VEL
LIN {X 0,Y 501.755,Z 401.913,A -85,B 0,C 180,E1 -12744.346,E2 -12744.346} C_VEL
LIN {X 0,Y 491.24,Z 387.337,A -85,B 0,C 180,E1 -12746.453,E2 -12746.453} C_VEL
LIN {X 0,Y 486.648,Z 381.318,A -85,B 0,C 180,E1 -12747.431,E2 -12747.431} C_VEL
LIN {X 0,Y 482.067,Z 375.33,A -85,B 0,C 180,E1 -12748.452,E2 -12748.452} C_VEL
LIN {X 0,Y 476.7,Z 368.155,A -85,B 0,C 180,E1 -12749.774,E2 -12749.774} C_VEL
LIN {X 0,Y 475.838,Z 366.288,A -85,B 0,C 180,E1 -12750.27,E2 -12750.27} C_VEL
LIN {X 0,Y 474.31,Z 363.181,A -85,B 0,C 180,E1 -12751.134,E2 -12751.134} C_VEL
LIN {X 0,Y 474.106,Z 362.155,A -85,B 0,C 180,E1 -12751.396,E2 -12751.396} C_VEL
LIN {X 0,Y 474.099,Z 362.157,A -85,B 0,C 180,E1 -12755.078,E2 -12755.078} C_VEL
LIN {X 0,Y 474.058,Z 362.173,A -85,B 0,C 180,E1 -12758.469,E2 -12758.469} C_VEL
LIN {X 0,Y 474.062,Z 362.178,A -85,B 0,C 180,E1 -12762.192,E2 -12762.192} C_VEL
LIN {X 0,Y 474.097,Z 362.173,A -85,B 0,C 180,E1 -12765.714,E2 -12765.714} C_VEL
LIN {X 0,Y 474.101,Z 362.157,A -85,B 0,C 180,E1 -12769.359,E2 -12769.359} C_VEL
LIN {X 0,Y 474.059,Z 362.149,A -85,B 0,C 180,E1 -12772.851,E2 -12772.851} C_VEL
LIN {X 0,Y 474.058,Z 362.159,A -85,B 0,C 180,E1 -12776.493,E2 -12776.493} C_VEL
LIN {X 0,Y 474.094,Z 362.175,A -85,B 0,C 180,E1 -12780,E2 -12780} C_VEL
LIN {X 0,Y 474.103,Z 362.165,A -85,B 0,C 180,E1 -12783.628,E2 -12783.628} C_VEL
LIN {X 0,Y 474.062,Z 362.15,A -85,B 0,C 180,E1 -12787.149,E2 -12787.149} C_VEL
LIN {X 0,Y 474.059,Z 362.155,A -85,B 0,C 180,E1 -12790.697,E2 -12790.697} C_VEL
LIN {X 0,Y 474.104,Z 362.17,A -85,B 0,C 180,E1 -12794.161,E2 -12794.161} C_VEL
LIN {X 0,Y 474.104,Z 362.174,A -85,B 0,C 180,E1 -12797.807,E2 -12797.807} C_VEL
LIN {X 0,Y 474.064,Z 362.166,A -85,B 0,C 180,E1 -12801.271,E2 -12801.271} C_VEL
LIN {X 0,Y 474.062,Z 362.162,A -85,B 0,C 180,E1 -12804.951,E2 -12804.951} C_VEL
LIN {X 0,Y 474.099,Z 362.155,A -85,B 0,C 180,E1 -12808.466,E2 -12808.466} C_VEL
LIN {X 0,Y 474.13,Z 362.33,A -85,B 0,C 180,E1 -12809.997,E2 -12809.997} C_VEL
LIN {X 0,Y 475.16,Z 365.223,A -85,B 0,C 180,E1 -12810.299,E2 -12810.299} C_VEL
LIN {X 0,Y 477.541,Z 367.806,A -85,B 0,C 180,E1 -12810.863,E2 -12810.863} C_VEL
LIN {X 0,Y 479.084,Z 368.962,A -85,B 0,C 180,E1 -12811.206,E2 -12811.206} C_VEL
LIN {X 0,Y 481.424,Z 372.644,A -85,B 0,C 180,E1 -12811.77,E2 -12811.77} C_VEL
LIN {X 0,Y 484.003,Z 375.105,A -85,B 0,C 180,E1 -12812.331,E2 -12812.331} C_VEL
LIN {X 0,Y 487,Z 379.202,A -85,B 0,C 180,E1 -12812.998,E2 -12812.998} C_VEL
LIN {X 0,Y 488.847,Z 381.091,A -85,B 0,C 180,E1 -12813.382,E2 -12813.382} C_VEL
LIN {X 0,Y 492.394,Z 385.584,A -85,B 0,C 180,E1 -12814.123,E2 -12814.123} C_VEL
LIN {X 0,Y 498.663,Z 393.693,A -85,B 0,C 180,E1 -12815.379,E2 -12815.379} C_VEL
LIN {X 0,Y 505.54,Z 402.521,A -85,B 0,C 180,E1 -12816.678,E2 -12816.678} C_VEL
LIN {X 0,Y 517.362,Z 418.732,A -85,B 0,C 180,E1 -12818.769,E2 -12818.769} C_VEL
LIN {X 0,Y 528.096,Z 434.552,A -85,B 0,C 180,E1 -12820.535,E2 -12820.535} C_VEL
LIN {X 0,Y 536.537,Z 448.782,A -85,B 0,C 180,E1 -12821.867,E2 -12821.867} C_VEL
LIN {X 0,Y 526.79,Z 699.598,A -85,B 0,C 180,E1 -12825.582,E2 -12825.582} C_VEL
LIN {X 0,Y 524.802,Z 746.676,A -85,B 0,C 180,E1 -12826.308,E2 -12826.308} C_VEL
LIN {X 0,Y 522.809,Z 770.868,A -85,B 0,C 180,E1 -12826.86,E2 -12826.86} C_VEL
LIN {X 0,Y 520.337,Z 794.469,A -85,B 0,C 180,E1 -12827.569,E2 -12827.569} C_VEL
LIN {X 0,Y 517.258,Z 817.479,A -85,B 0,C 180,E1 -12828.468,E2 -12828.468} C_VEL
LIN {X 0,Y 514.167,Z 837.672,A -85,B 0,C 180,E1 -12829.421,E2 -12829.421} C_VEL
LIN {X 0,Y 510.073,Z 860.934,A -85,B 0,C 180,E1 -12830.743,E2 -12830.743} C_VEL
LIN {X 0,Y 506.346,Z 880.144,A -85,B 0,C 180,E1 -12832.039,E2 -12832.039} C_VEL
LIN {X 0,Y 501.702,Z 902.128,A -85,B 0,C 180,E1 -12833.778,E2 -12833.778} C_VEL
LIN {X 0,Y 497.694,Z 919.895,A -85,B 0,C 180,E1 -12835.42,E2 -12835.42} C_VEL
LIN {X 0,Y 493.167,Z 939.362,A -85,B 0,C 180,E1 -12837.505,E2 -12837.505} C_VEL
LIN {X 0,Y 489.483,Z 954.808,A -85,B 0,C 180,E1 -12839.427,E2 -12839.427} C_VEL
LIN {X 0,Y 485.637,Z 971.077,A -85,B 0,C 180,E1 -12841.735,E2 -12841.735} C_VEL
LIN {X 0,Y 482.268,Z 985.493,A -85,B 0,C 180,E1 -12844.135,E2 -12844.135} C_VEL
LIN {X 0,Y 482.108,Z 986.206,A -85,B 0,C 180,E1 -12844.261,E2 -12844.261} C_VEL
LIN {X 0,Y 480.224,Z 990.593,A -85,B 0,C 180,E1 -12844.996,E2 -12844.996} C_VEL
LIN {X 0,Y 472.247,Z 1001.226,A -85,B 0,C 180,E1 -12846.816,E2 -12846.816} C_VEL
LIN {X 0,Y 470.474,Z 1005.023,A -85,B 0,C 180,E1 -12847.606,E2 -12847.606} C_VEL
LIN {X 0,Y 468.081,Z 1016.786,A -85,B 0,C 180,E1 -12850.535,E2 -12850.535} C_VEL
LIN {X 0,Y 466.554,Z 1025.315,A -85,B 0,C 180,E1 -12853.054,E2 -12853.054} C_VEL
LIN {X 0,Y 465.304,Z 1033.84,A -85,B 0,C 180,E1 -12856.074,E2 -12856.074} C_VEL
LIN {X 0,Y 464.588,Z 1039.988,A -85,B 0,C 180,E1 -12858.831,E2 -12858.831} C_VEL
LIN {X 0,Y 464.184,Z 1045.014,A -85,B 0,C 180,E1 -12861.702,E2 -12861.702} C_VEL
LIN {X 0,Y 464,Z 1048.467,A -85,B 0,C 180,E1 -12864.615,E2 -12864.615} C_VEL
LIN {X 0,Y 463.95,Z 1050.246,A -85,B 0,C 180,E1 -12867.035,E2 -12867.035} C_VEL
LIN {X 0,Y 463.935,Z 1051.079,A -85,B 0,C 180,E1 -12869.753,E2 -12869.753} C_VEL
LIN {X 0,Y 463.946,Z 1050.43,A -85,B 0,C 180,E1 -12872.718,E2 -12872.718} C_VEL
LIN {X 0,Y 463.994,Z 1048.724,A -85,B 0,C 180,E1 -12875.193,E2 -12875.193} C_VEL
LIN {X 0,Y 464.123,Z 1045.808,A -85,B 0,C 180,E1 -12877.801,E2 -12877.801} C_VEL
LIN {X 0,Y 464.527,Z 1040.673,A -85,B 0,C 180,E1 -12880.919,E2 -12880.919} C_VEL
LIN {X 0,Y 465.158,Z 1034.955,A -85,B 0,C 180,E1 -12883.551,E2 -12883.551} C_VEL
LIN {X 0,Y 466.341,Z 1026.773,A -85,B 0,C 180,E1 -12886.579,E2 -12886.579} C_VEL
LIN {X 0,Y 467.851,Z 1018.017,A -85,B 0,C 180,E1 -12889.216,E2 -12889.216} C_VEL
LIN {X 0,Y 470.019,Z 1007.257,A -85,B 0,C 180,E1 -12891.988,E2 -12891.988} C_VEL
LIN {X 0,Y 472.708,Z 994.999,A -85,B 0,C 180,E1 -12894.627,E2 -12894.627} C_VEL
LIN {X 0,Y 475.896,Z 981.655,A -85,B 0,C 180,E1 -12897.125,E2 -12897.125} C_VEL
LIN {X 0,Y 479.493,Z 966.935,A -85,B 0,C 180,E1 -12899.481,E2 -12899.481} C_VEL
LIN {X 0,Y 483.204,Z 952.01,A -85,B 0,C 180,E1 -12901.569,E2 -12901.569} C_VEL
LIN {X 0,Y 487.828,Z 933.406,A -85,B 0,C 180,E1 -12903.813,E2 -12903.813} C_VEL
LIN {X 0,Y 491.702,Z 917.337,A -85,B 0,C 180,E1 -12905.491,E2 -12905.491} C_VEL
LIN {X 0,Y 496.209,Z 898.005,A -85,B 0,C 180,E1 -12907.255,E2 -12907.255} C_VEL
LIN {X 0,Y 500.441,Z 878.25,A -85,B 0,C 180,E1 -12908.784,E2 -12908.784} C_VEL
LIN {X 0,Y 504.582,Z 857.553,A -85,B 0,C 180,E1 -12910.167,E2 -12910.167} C_VEL
LIN {X 0,Y 508.6,Z 834.912,A -85,B 0,C 180,E1 -12911.418,E2 -12911.418} C_VEL
LIN {X 0,Y 511.962,Z 813.375,A -85,B 0,C 180,E1 -12912.417,E2 -12912.417} C_VEL
LIN {X 0,Y 515.108,Z 789.117,A -85,B 0,C 180,E1 -12913.313,E2 -12913.313} C_VEL
LIN {X 0,Y 517.437,Z 767.109,A -85,B 0,C 180,E1 -12913.95,E2 -12913.95} C_VEL
LIN {X 0,Y 519.406,Z 741.24,A -85,B 0,C 180,E1 -12914.495,E2 -12914.495} C_VEL
LIN {X 0,Y 528.678,Z 511.734,A -85,B 0,C 180,E1 -12917.937,E2 -12917.937} C_VEL
LIN {X 0,Y 531.032,Z 452.011,A -85,B 0,C 180,E1 -12918.846,E2 -12918.846} C_VEL
LIN {X 0,Y 520.887,Z 435.422,A -85,B 0,C 180,E1 -12920.5,E2 -12920.5} C_VEL
LIN {X 0,Y 508.323,Z 417.281,A -85,B 0,C 180,E1 -12922.674,E2 -12922.674} C_VEL
LIN {X 0,Y 497.125,Z 402.397,A -85,B 0,C 180,E1 -12924.777,E2 -12924.777} C_VEL
LIN {X 0,Y 488.908,Z 391.902,A -85,B 0,C 180,E1 -12926.447,E2 -12926.447} C_VEL
LIN {X 0,Y 484.814,Z 386.762,A -85,B 0,C 180,E1 -12927.327,E2 -12927.327} C_VEL
LIN {X 0,Y 481.289,Z 382.317,A -85,B 0,C 180,E1 -12928.115,E2 -12928.115} C_VEL
LIN {X 0,Y 477.012,Z 377.363,A -85,B 0,C 180,E1 -12929.099,E2 -12929.099} C_VEL
LIN {X 0,Y 475.922,Z 375.639,A -85,B 0,C 180,E1 -12929.371,E2 -12929.371} C_VEL
LIN {X 0,Y 472.834,Z 372.722,A -85,B 0,C 180,E1 -12930.1,E2 -12930.1} C_VEL
LIN {X 0,Y 471.086,Z 369.606,A -85,B 0,C 180,E1 -12930.57,E2 -12930.57} C_VEL
LIN {X 0,Y 468.056,Z 367.442,A -85,B 0,C 180,E1 -12931.306,E2 -12931.306} C_VEL
LIN {X 0,Y 466.483,Z 364.56,A -85,B 0,C 180,E1 -12931.756,E2 -12931.756} C_VEL
LIN {X 0,Y 466.177,Z 363.142,A -85,B 0,C 180,E1 -12931.883,E2 -12931.883} C_VEL
LIN {X 0,Y 466.145,Z 363.146,A -85,B 0,C 180,E1 -12935.544,E2 -12935.544} C_VEL
LIN {X 0,Y 466.117,Z 363.158,A -85,B 0,C 180,E1 -12939.008,E2 -12939.008} C_VEL
LIN {X 0,Y 466.127,Z 363.168,A -85,B 0,C 180,E1 -12942.663,E2 -12942.663} C_VEL
LIN {X 0,Y 466.167,Z 363.155,A -85,B 0,C 180,E1 -12946.226,E2 -12946.226} C_VEL
LIN {X 0,Y 466.152,Z 363.139,A -85,B 0,C 180,E1 -12949.915,E2 -12949.915} C_VEL
LIN {X 0,Y 466.114,Z 363.141,A -85,B 0,C 180,E1 -12953.348,E2 -12953.348} C_VEL
LIN {X 0,Y 466.118,Z 363.156,A -85,B 0,C 180,E1 -12957.049,E2 -12957.049} C_VEL
LIN {X 0,Y 466.154,Z 363.167,A -85,B 0,C 180,E1 -12960.615,E2 -12960.615} C_VEL
LIN {X 0,Y 466.16,Z 363.143,A -85,B 0,C 180,E1 -12964.305,E2 -12964.305} C_VEL
LIN {X 0,Y 466.12,Z 363.139,A -85,B 0,C 180,E1 -12967.767,E2 -12967.767} C_VEL
LIN {X 0,Y 466.115,Z 363.148,A -85,B 0,C 180,E1 -12971.382,E2 -12971.382} C_VEL
LIN {X 0,Y 466.147,Z 363.162,A -85,B 0,C 180,E1 -12974.916,E2 -12974.916} C_VEL
LIN {X 0,Y 466.166,Z 363.161,A -85,B 0,C 180,E1 -12978.548,E2 -12978.548} C_VEL
LIN {X 0,Y 466.126,Z 363.156,A -85,B 0,C 180,E1 -12982.076,E2 -12982.076} C_VEL
LIN {X 0,Y 466.117,Z 363.157,A -85,B 0,C 180,E1 -12985.715,E2 -12985.715} C_VEL
LIN {X 0,Y 466.166,Z 363.255,A -85,B 0,C 180,E1 -12987.047,E2 -12987.047} C_VEL
LIN {X 0,Y 467.351,Z 366.527,A -85,B 0,C 180,E1 -12987.94,E2 -12987.94} C_VEL
LIN {X 0,Y 468.727,Z 368.434,A -85,B 0,C 180,E1 -12988.544,E2 -12988.544} C_VEL
LIN {X 0,Y 471.679,Z 372.636,A -85,B 0,C 180,E1 -12989.32,E2 -12989.32} C_VEL
LIN {X 0,Y 474.216,Z 375.639,A -85,B 0,C 180,E1 -12989.947,E2 -12989.947} C_VEL
LIN {X 0,Y 481.916,Z 385.712,A -85,B 0,C 180,E1 -12991.769,E2 -12991.769} C_VEL
LIN {X 0,Y 486.526,Z 391.95,A -85,B 0,C 180,E1 -12992.795,E2 -12992.795} C_VEL
LIN {X 0,Y 492.722,Z 400.378,A -85,B 0,C 180,E1 -12994.105,E2 -12994.105} C_VEL
LIN {X 0,Y 503.954,Z 416.536,A -85,B 0,C 180,E1 -12996.317,E2 -12996.317} C_VEL
LIN {X 0,Y 515.203,Z 434.005,A -85,B 0,C 180,E1 -12998.361,E2 -12998.361} C_VEL
LIN {X 0,Y 526.717,Z 453.256,A -85,B 0,C 180,E1 -13000.306,E2 -13000.306} C_VEL
LIN {X 0,Y 531,Z 461.211,A -85,B 0,C 180,E1 -13001.005,E2 -13001.005} C_VEL
LIN {X 0,Y 521.039,Z 709.765,A -85,B 0,C 180,E1 -13004.715,E2 -13004.715} C_VEL
LIN {X 0,Y 518.683,Z 765.45,A -85,B 0,C 180,E1 -13005.572,E2 -13005.572} C_VEL
LIN {X 0,Y 516.518,Z 790.202,A -85,B 0,C 180,E1 -13006.115,E2 -13006.115} C_VEL
LIN {X 0,Y 514.164,Z 810.979,A -85,B 0,C 180,E1 -13006.715,E2 -13006.715} C_VEL
LIN {X 0,Y 510.839,Z 834.994,A -85,B 0,C 180,E1 -13007.6,E2 -13007.6} C_VEL
LIN {X 0,Y 507.699,Z 854.567,A -85,B 0,C 180,E1 -13008.492,E2 -13008.492} C_VEL
LIN {X 0,Y 503.76,Z 876.603,A -85,B 0,C 180,E1 -13009.679,E2 -13009.679} C_VEL
LIN {X 0,Y 499.494,Z 897.727,A -85,B 0,C 180,E1 -13011.055,E2 -13011.055} C_VEL
LIN {X 0,Y 495.363,Z 916.993,A -85,B 0,C 180,E1 -13012.513,E2 -13012.513} C_VEL
LIN {X 0,Y 490.635,Z 937.676,A -85,B 0,C 180,E1 -13014.348,E2 -13014.348} C_VEL
LIN {X 0,Y 486.754,Z 954.094,A -85,B 0,C 180,E1 -13016.031,E2 -13016.031} C_VEL
LIN {X 0,Y 482.297,Z 972.719,A -85,B 0,C 180,E1 -13018.225,E2 -13018.225} C_VEL
LIN {X 0,Y 478.583,Z 988.054,A -85,B 0,C 180,E1 -13020.32,E2 -13020.32} C_VEL
LIN {X 0,Y 475.058,Z 1003.286,A -85,B 0,C 180,E1 -13022.688,E2 -13022.688} C_VEL
LIN {X 0,Y 471.808,Z 1017.699,A -85,B 0,C 180,E1 -13025.323,E2 -13025.323} C_VEL
LIN {X 0,Y 469.257,Z 1030.316,A -85,B 0,C 180,E1 -13027.974,E2 -13027.974} C_VEL
LIN {X 0,Y 467.221,Z 1041.424,A -85,B 0,C 180,E1 -13030.757,E2 -13030.757} C_VEL
LIN {X 0,Y 465.783,Z 1050.922,A -85,B 0,C 180,E1 -13033.539,E2 -13033.539} C_VEL
LIN {X 0,Y 464.793,Z 1059.131,A -85,B 0,C 180,E1 -13036.501,E2 -13036.501} C_VEL
LIN {X 0,Y 464.291,Z 1064.924,A -85,B 0,C 180,E1 -13039.075,E2 -13039.075} C_VEL
LIN {X 0,Y 464.002,Z 1070.13,A -85,B 0,C 180,E1 -13042.073,E2 -13042.073} C_VEL
LIN {X 0,Y 463.944,Z 1073.239,A -85,B 0,C 180,E1 -13044.689,E2 -13044.689} C_VEL
LIN {X 0,Y 463.936,Z 1075.074,A -85,B 0,C 180,E1 -13047.159,E2 -13047.159} C_VEL
LIN {X 0,Y 463.946,Z 1075.892,A -85,B 0,C 180,E1 -13050,E2 -13050} C_VEL
LIN {X 0,Y 463.936,Z 1075.072,A -85,B 0,C 180,E1 -13052.841,E2 -13052.841} C_VEL
LIN {X 0,Y 463.943,Z 1073.229,A -85,B 0,C 180,E1 -13055.317,E2 -13055.317} C_VEL
LIN {X 0,Y 464.023,Z 1069.798,A -85,B 0,C 180,E1 -13058.176,E2 -13058.176} C_VEL
LIN {X 0,Y 464.31,Z 1064.66,A -85,B 0,C 180,E1 -13061.05,E2 -13061.05} C_VEL
LIN {X 0,Y 464.808,Z 1058.97,A -85,B 0,C 180,E1 -13063.561,E2 -13063.561} C_VEL
LIN {X 0,Y 465.835,Z 1050.497,A -85,B 0,C 180,E1 -13066.587,E2 -13066.587} C_VEL
LIN {X 0,Y 467.219,Z 1041.413,A -85,B 0,C 180,E1 -13069.243,E2 -13069.243} C_VEL
LIN {X 0,Y 469.276,Z 1030.196,A -85,B 0,C 180,E1 -13072.049,E2 -13072.049} C_VEL
LIN {X 0,Y 471.804,Z 1017.677,A -85,B 0,C 180,E1 -13074.677,E2 -13074.677} C_VEL
LIN {X 0,Y 475.052,Z 1003.253,A -85,B 0,C 180,E1 -13077.313,E2 -13077.313} C_VEL
LIN {X 0,Y 478.575,Z 988.012,A -85,B 0,C 180,E1 -13079.681,E2 -13079.681} C_VEL
LIN {X 0,Y 482.527,Z 971.736,A -85,B 0,C 180,E1 -13081.898,E2 -13081.898} C_VEL
LIN {X 0,Y 486.899,Z 953.366,A -85,B 0,C 180,E1 -13084.041,E2 -13084.041} C_VEL
LIN {X 0,Y 491.078,Z 935.696,A -85,B 0,C 180,E1 -13085.837,E2 -13085.837} C_VEL
LIN {X 0,Y 495.833,Z 914.671,A -85,B 0,C 180,E1 -13087.664,E2 -13087.664} C_VEL
LIN {X 0,Y 499.829,Z 895.979,A -85,B 0,C 180,E1 -13089.061,E2 -13089.061} C_VEL
LIN {X 0,Y 504.289,Z 873.434,A -85,B 0,C 180,E1 -13090.493,E2 -13090.493} C_VEL
LIN {X 0,Y 507.873,Z 853.266,A -85,B 0,C 180,E1 -13091.566,E2 -13091.566} C_VEL
LIN {X 0,Y 511.448,Z 830.879,A -85,B 0,C 180,E1 -13092.566,E2 -13092.566} C_VEL
LIN {X 0,Y 514.494,Z 807.796,A -85,B 0,C 180,E1 -13093.378,E2 -13093.378} C_VEL
LIN {X 0,Y 516.832,Z 786.765,A -85,B 0,C 180,E1 -13093.965,E2 -13093.965} C_VEL
LIN {X 0,Y 518.874,Z 760.812,A -85,B 0,C 180,E1 -13094.499,E2 -13094.499} C_VEL
LIN {X 0,Y 527.888,Z 534.597,A -85,B 0,C 180,E1 -13097.892,E2 -13097.892} C_VEL
LIN {X 0,Y 530.862,Z 460.745,A -85,B 0,C 180,E1 -13099.005,E2 -13099.005} C_VEL
LIN {X 0,Y 518.969,Z 440.26,A -85,B 0,C 180,E1 -13100.965,E2 -13100.965} C_VEL
LIN {X 0,Y 508.163,Z 423.037,A -85,B 0,C 180,E1 -13102.873,E2 -13102.873} C_VEL
LIN {X 0,Y 498.075,Z 407.971,A -85,B 0,C 180,E1 -13104.788,E2 -13104.788} C_VEL
LIN {X 0,Y 488.199,Z 394.073,A -85,B 0,C 180,E1 -13106.814,E2 -13106.814} C_VEL
LIN {X 0,Y 479.367,Z 382.342,A -85,B 0,C 180,E1 -13108.779,E2 -13108.779} C_VEL
LIN {X 0,Y 472.092,Z 373.049,A -85,B 0,C 180,E1 -13110.534,E2 -13110.534} C_VEL
LIN {X 0,Y 468.987,Z 368.945,A -85,B 0,C 180,E1 -13111.334,E2 -13111.334} C_VEL
LIN {X 0,Y 468.223,Z 367.602,A -85,B 0,C 180,E1 -13111.621,E2 -13111.621} C_VEL
LIN {X 0,Y 466.473,Z 364.68,A -85,B 0,C 180,E1 -13112.558,E2 -13112.558} C_VEL
LIN {X 0,Y 466.152,Z 363.142,A -85,B 0,C 180,E1 -13112.952,E2 -13112.952} C_VEL
LIN {X 0,Y 466.119,Z 363.147,A -85,B 0,C 180,E1 -13116.484,E2 -13116.484} C_VEL
LIN {X 0,Y 466.117,Z 363.145,A -85,B 0,C 180,E1 -13120.188,E2 -13120.188} C_VEL
LIN {X 0,Y 466.154,Z 363.138,A -85,B 0,C 180,E1 -13123.68,E2 -13123.68} C_VEL
LIN {X 0,Y 466.146,Z 363.149,A -85,B 0,C 180,E1 -13127.11,E2 -13127.11} C_VEL
LIN {X 0,Y 466.121,Z 363.169,A -85,B 0,C 180,E1 -13130.665,E2 -13130.665} C_VEL
LIN {X 0,Y 466.124,Z 363.158,A -85,B 0,C 180,E1 -13134.337,E2 -13134.337} C_VEL
LIN {X 0,Y 466.154,Z 363.137,A -85,B 0,C 180,E1 -13137.91,E2 -13137.91} C_VEL
LIN {X 0,Y 466.145,Z 363.141,A -85,B 0,C 180,E1 -13141.352,E2 -13141.352} C_VEL
LIN {X 0,Y 466.121,Z 363.167,A -85,B 0,C 180,E1 -13144.922,E2 -13144.922} C_VEL
LIN {X 0,Y 466.123,Z 363.165,A -85,B 0,C 180,E1 -13148.636,E2 -13148.636} C_VEL
LIN {X 0,Y 466.158,Z 363.139,A -85,B 0,C 180,E1 -13152.134,E2 -13152.134} C_VEL
LIN {X 0,Y 466.155,Z 363.137,A -85,B 0,C 180,E1 -13155.68,E2 -13155.68} C_VEL
LIN {X 0,Y 466.124,Z 363.15,A -85,B 0,C 180,E1 -13159.16,E2 -13159.16} C_VEL
LIN {X 0,Y 466.126,Z 363.158,A -85,B 0,C 180,E1 -13162.847,E2 -13162.847} C_VEL
LIN {X 0,Y 466.164,Z 363.161,A -85,B 0,C 180,E1 -13166.36,E2 -13166.36} C_VEL
LIN {X 0,Y 466.194,Z 363.279,A -85,B 0,C 180,E1 -13168.277,E2 -13168.277} C_VEL
LIN {X 0,Y 467.23,Z 366.28,A -85,B 0,C 180,E1 -13168.609,E2 -13168.609} C_VEL
LIN {X 0,Y 469.713,Z 368.887,A -85,B 0,C 180,E1 -13169.245,E2 -13169.245} C_VEL
LIN {X 0,Y 471.307,Z 369.95,A -85,B 0,C 180,E1 -13169.625,E2 -13169.625} C_VEL
LIN {X 0,Y 473.52,Z 373.604,A -85,B 0,C 180,E1 -13170.205,E2 -13170.205} C_VEL
LIN {X 0,Y 476.393,Z 376.275,A -85,B 0,C 180,E1 -13170.876,E2 -13170.876} C_VEL
LIN {X 0,Y 479.44,Z 380.387,A -85,B 0,C 180,E1 -13171.601,E2 -13171.601} C_VEL
LIN {X 0,Y 481.326,Z 382.399,A -85,B 0,C 180,E1 -13172.022,E2 -13172.022} C_VEL
LIN {X 0,Y 484.866,Z 386.809,A -85,B 0,C 180,E1 -13172.809,E2 -13172.809} C_VEL
LIN {X 0,Y 491.301,Z 394.969,A -85,B 0,C 180,E1 -13174.175,E2 -13174.175} C_VEL
LIN {X 0,Y 499.509,Z 405.516,A -85,B 0,C 180,E1 -13175.804,E2 -13175.804} C_VEL
LIN {X 0,Y 509.614,Z 419.265,A -85,B 0,C 180,E1 -13177.675,E2 -13177.675} C_VEL
LIN {X 0,Y 521.51,Z 436.368,A -85,B 0,C 180,E1 -13179.713,E2 -13179.713} C_VEL
LIN {X 0,Y 531.092,Z 452.303,A -85,B 0,C 180,E1 -13181.273,E2 -13181.273} C_VEL
LIN {X 0,Y 520.938,Z 704.158,A -85,B 0,C 180,E1 -13185.031,E2 -13185.031} C_VEL
LIN {X 0,Y 519.007,Z 747.432,A -85,B 0,C 180,E1 -13185.708,E2 -13185.708} C_VEL
LIN {X 0,Y 516.964,Z 771.356,A -85,B 0,C 180,E1 -13186.259,E2 -13186.259} C_VEL
LIN {X 0,Y 514.395,Z 795.08,A -85,B 0,C 180,E1 -13186.978,E2 -13186.978} C_VEL
LIN {X 0,Y 511.257,Z 817.703,A -85,B 0,C 180,E1 -13187.87,E2 -13187.87} C_VEL
LIN {X 0,Y 508.065,Z 837.895,A -85,B 0,C 180,E1 -13188.829,E2 -13188.829} C_VEL
LIN {X 0,Y 503.894,Z 860.815,A -85,B 0,C 180,E1 -13190.138,E2 -13190.138} C_VEL
LIN {X 0,Y 500.089,Z 879.773,A -85,B 0,C 180,E1 -13191.424,E2 -13191.424} C_VEL
LIN {X 0,Y 495.473,Z 901.025,A -85,B 0,C 180,E1 -13193.104,E2 -13193.104} C_VEL
LIN {X 0,Y 491.288,Z 918.91,A -85,B 0,C 180,E1 -13194.761,E2 -13194.761} C_VEL
LIN {X 0,Y 486.807,Z 937.547,A -85,B 0,C 180,E1 -13196.742,E2 -13196.742} C_VEL
LIN {X 0,Y 482.603,Z 954.322,A -85,B 0,C 180,E1 -13198.836,E2 -13198.836} C_VEL
LIN {X 0,Y 478.619,Z 970.52,A -85,B 0,C 180,E1 -13201.146,E2 -13201.146} C_VEL
LIN {X 0,Y 474.976,Z 985.313,A -85,B 0,C 180,E1 -13203.629,E2 -13203.629} C_VEL
LIN {X 0,Y 471.973,Z 998.312,A -85,B 0,C 180,E1 -13206.132,E2 -13206.132} C_VEL
LIN {X 0,Y 470.474,Z 1005.023,A -85,B 0,C 180,E1 -13207.606,E2 -13207.606} C_VEL
LIN {X 0,Y 468.74,Z 1008.746,A -85,B 0,C 180,E1 -13208.412,E2 -13208.412} C_VEL
LIN {X 0,Y 460.837,Z 1018.143,A -85,B 0,C 180,E1 -13210.552,E2 -13210.552} C_VEL
LIN {X 0,Y 459.61,Z 1020.875,A -85,B 0,C 180,E1 -13211.292,E2 -13211.292} C_VEL
LIN {X 0,Y 457.987,Z 1030.091,A -85,B 0,C 180,E1 -13214.325,E2 -13214.325} C_VEL
LIN {X 0,Y 457.047,Z 1036.738,A -85,B 0,C 180,E1 -13216.978,E2 -13216.978} C_VEL
LIN {X 0,Y 456.381,Z 1043.001,A -85,B 0,C 180,E1 -13220.16,E2 -13220.16} C_VEL
LIN {X 0,Y 456.108,Z 1046.843,A -85,B 0,C 180,E1 -13222.822,E2 -13222.822} C_VEL
LIN {X 0,Y 455.987,Z 1049.634,A -85,B 0,C 180,E1 -13225.598,E2 -13225.598} C_VEL
LIN {X 0,Y 455.942,Z 1051.092,A -85,B 0,C 180,E1 -13228.618,E2 -13228.618} C_VEL
LIN {X 0,Y 455.949,Z 1051.152,A -85,B 0,C 180,E1 -13231.131,E2 -13231.131} C_VEL
LIN {X 0,Y 455.971,Z 1050.08,A -85,B 0,C 180,E1 -13233.83,E2 -13233.83} C_VEL
LIN {X 0,Y 456.075,Z 1047.274,A -85,B 0,C 180,E1 -13236.926,E2 -13236.926} C_VEL
LIN {X 0,Y 456.327,Z 1043.554,A -85,B 0,C 180,E1 -13239.588,E2 -13239.588} C_VEL
LIN {X 0,Y 456.928,Z 1037.851,A -85,B 0,C 180,E1 -13242.64,E2 -13242.64} C_VEL
LIN {X 0,Y 457.855,Z 1030.957,A -85,B 0,C 180,E1 -13245.452,E2 -13245.452} C_VEL
LIN {X 0,Y 459.209,Z 1023.035,A -85,B 0,C 180,E1 -13248.142,E2 -13248.142} C_VEL
LIN {X 0,Y 461.287,Z 1012.552,A -85,B 0,C 180,E1 -13251.089,E2 -13251.089} C_VEL
LIN {X 0,Y 463.569,Z 1002.257,A -85,B 0,C 180,E1 -13253.551,E2 -13253.551} C_VEL
LIN {X 0,Y 466.846,Z 988.794,A -85,B 0,C 180,E1 -13256.318,E2 -13256.318} C_VEL
LIN {X 0,Y 470.088,Z 975.868,A -85,B 0,C 180,E1 -13258.593,E2 -13258.593} C_VEL
LIN {X 0,Y 474.142,Z 960.457,A -85,B 0,C 180,E1 -13260.968,E2 -13260.968} C_VEL
LIN {X 0,Y 478.5,Z 943.486,A -85,B 0,C 180,E1 -13263.195,E2 -13263.195} C_VEL
LIN {X 0,Y 483.012,Z 925.916,A -85,B 0,C 180,E1 -13265.207,E2 -13265.207} C_VEL
LIN {X 0,Y 487.675,Z 906.8,A -85,B 0,C 180,E1 -13267.07,E2 -13267.07} C_VEL
LIN {X 0,Y 491.923,Z 888.607,A -85,B 0,C 180,E1 -13268.61,E2 -13268.61} C_VEL
LIN {X 0,Y 496.617,Z 866.718,A -85,B 0,C 180,E1 -13270.188,E2 -13270.188} C_VEL
LIN {X 0,Y 500.244,Z 848.151,A -85,B 0,C 180,E1 -13271.325,E2 -13271.325} C_VEL
LIN {X 0,Y 504.206,Z 825.763,A -85,B 0,C 180,E1 -13272.489,E2 -13272.489} C_VEL
LIN {X 0,Y 507.401,Z 804.139,A -85,B 0,C 180,E1 -13273.403,E2 -13273.403} C_VEL
LIN {X 0,Y 510.094,Z 782.95,A -85,B 0,C 180,E1 -13274.134,E2 -13274.134} C_VEL
LIN {X 0,Y 512.557,Z 757.883,A -85,B 0,C 180,E1 -13274.792,E2 -13274.792} C_VEL
LIN {X 0,Y 514.014,Z 736.297,A -85,B 0,C 180,E1 -13275.207,E2 -13275.207} C_VEL
LIN {X 0,Y 524.457,Z 486.413,A -85,B 0,C 180,E1 -13278.969,E2 -13278.969} C_VEL
LIN {X 0,Y 525.642,Z 455.652,A -85,B 0,C 180,E1 -13279.452,E2 -13279.452} C_VEL
LIN {X 0,Y 516.802,Z 441.143,A -85,B 0,C 180,E1 -13280.931,E2 -13280.931} C_VEL
LIN {X 0,Y 504.708,Z 423.504,A -85,B 0,C 180,E1 -13283.074,E2 -13283.074} C_VEL
LIN {X 0,Y 493.764,Z 408.824,A -85,B 0,C 180,E1 -13285.176,E2 -13285.176} C_VEL
LIN {X 0,Y 485.767,Z 398.513,A -85,B 0,C 180,E1 -13286.837,E2 -13286.837} C_VEL
LIN {X 0,Y 481.718,Z 393.434,A -85,B 0,C 180,E1 -13287.726,E2 -13287.726} C_VEL
LIN {X 0,Y 477.194,Z 387.841,A -85,B 0,C 180,E1 -13288.761,E2 -13288.761} C_VEL
LIN {X 0,Y 473.712,Z 383.395,A -85,B 0,C 180,E1 -13289.598,E2 -13289.598} C_VEL
LIN {X 0,Y 469.715,Z 378.998,A -85,B 0,C 180,E1 -13290.58,E2 -13290.58} C_VEL
LIN {X 0,Y 468.365,Z 376.856,A -85,B 0,C 180,E1 -13290.943,E2 -13290.943} C_VEL
LIN {X 0,Y 465.207,Z 374.065,A -85,B 0,C 180,E1 -13291.745,E2 -13291.745} C_VEL
LIN {X 0,Y 463.14,Z 370.563,A -85,B 0,C 180,E1 -13292.343,E2 -13292.343} C_VEL
LIN {X 0,Y 460.076,Z 368.388,A -85,B 0,C 180,E1 -13293.16,E2 -13293.16} C_VEL
LIN {X 0,Y 458.532,Z 365.577,A -85,B 0,C 180,E1 -13293.644,E2 -13293.644} C_VEL
LIN {X 0,Y 458.227,Z 364.141,A -85,B 0,C 180,E1 -13293.776,E2 -13293.776} C_VEL
LIN {X 0,Y 458.195,Z 364.14,A -85,B 0,C 180,E1 -13297.414,E2 -13297.414} C_VEL
LIN {X 0,Y 458.178,Z 364.134,A -85,B 0,C 180,E1 -13301.024,E2 -13301.024} C_VEL
LIN {X 0,Y 458.184,Z 364.127,A -85,B 0,C 180,E1 -13304.703,E2 -13304.703} C_VEL
LIN {X 0,Y 458.225,Z 364.129,A -85,B 0,C 180,E1 -13308.164,E2 -13308.164} C_VEL
LIN {X 0,Y 458.208,Z 364.151,A -85,B 0,C 180,E1 -13311.846,E2 -13311.846} C_VEL
LIN {X 0,Y 458.177,Z 364.15,A -85,B 0,C 180,E1 -13315.369,E2 -13315.369} C_VEL
LIN {X 0,Y 458.177,Z 364.131,A -85,B 0,C 180,E1 -13319.125,E2 -13319.125} C_VEL
LIN {X 0,Y 458.209,Z 364.124,A -85,B 0,C 180,E1 -13322.627,E2 -13322.627} C_VEL
LIN {X 0,Y 458.234,Z 364.137,A -85,B 0,C 180,E1 -13326.389,E2 -13326.389} C_VEL
LIN {X 0,Y 458.199,Z 364.158,A -85,B 0,C 180,E1 -13330.054,E2 -13330.054} C_VEL
LIN {X 0,Y 458.176,Z 364.144,A -85,B 0,C 180,E1 -13333.632,E2 -13333.632} C_VEL
LIN {X 0,Y 458.183,Z 364.131,A -85,B 0,C 180,E1 -13337.265,E2 -13337.265} C_VEL
LIN {X 0,Y 458.224,Z 364.124,A -85,B 0,C 180,E1 -13340.835,E2 -13340.835} C_VEL
LIN {X 0,Y 458.203,Z 364.129,A -85,B 0,C 180,E1 -13344.358,E2 -13344.358} C_VEL
LIN {X 0,Y 458.197,Z 364.199,A -85,B 0,C 180,E1 -13345.323,E2 -13345.323} C_VEL
LIN {X 0,Y 459.634,Z 367.818,A -85,B 0,C 180,E1 -13346.38,E2 -13346.38} C_VEL
LIN {X 0,Y 461.732,Z 370.304,A -85,B 0,C 180,E1 -13346.98,E2 -13346.98} C_VEL
LIN {X 0,Y 465.001,Z 374.317,A -85,B 0,C 180,E1 -13347.885,E2 -13347.885} C_VEL
LIN {X 0,Y 466.364,Z 375.923,A -85,B 0,C 180,E1 -13348.248,E2 -13348.248} C_VEL
LIN {X 0,Y 469.749,Z 380.337,A -85,B 0,C 180,E1 -13349.138,E2 -13349.138} C_VEL
LIN {X 0,Y 478.863,Z 392.276,A -85,B 0,C 180,E1 -13351.362,E2 -13351.362} C_VEL
LIN {X 0,Y 488.783,Z 405.821,A -85,B 0,C 180,E1 -13353.562,E2 -13353.562} C_VEL
LIN {X 0,Y 500.507,Z 422.949,A -85,B 0,C 180,E1 -13355.933,E2 -13355.933} C_VEL
LIN {X 0,Y 511.422,Z 440.087,A -85,B 0,C 180,E1 -13357.962,E2 -13357.962} C_VEL
LIN {X 0,Y 522.662,Z 459.112,A -85,B 0,C 180,E1 -13359.905,E2 -13359.905} C_VEL
LIN {X 0,Y 525.6,Z 464.718,A -85,B 0,C 180,E1 -13360.399,E2 -13360.399} C_VEL
LIN {X 0,Y 515.314,Z 712.225,A -85,B 0,C 180,E1 -13364.121,E2 -13364.121} C_VEL
LIN {X 0,Y 512.956,Z 765.684,A -85,B 0,C 180,E1 -13364.951,E2 -13364.951} C_VEL
LIN {X 0,Y 510.726,Z 790.247,A -85,B 0,C 180,E1 -13365.496,E2 -13365.496} C_VEL
LIN {X 0,Y 508.286,Z 811.1,A -85,B 0,C 180,E1 -13366.102,E2 -13366.102} C_VEL
LIN {X 0,Y 504.683,Z 836.074,A -85,B 0,C 180,E1 -13367.036,E2 -13367.036} C_VEL
LIN {X 0,Y 501.451,Z 855.492,A -85,B 0,C 180,E1 -13367.934,E2 -13367.934} C_VEL
LIN {X 0,Y 497.389,Z 877.347,A -85,B 0,C 180,E1 -13369.13,E2 -13369.13} C_VEL
LIN {X 0,Y 492.92,Z 898.624,A -85,B 0,C 180,E1 -13370.538,E2 -13370.538} C_VEL
LIN {X 0,Y 488.278,Z 919.504,A -85,B 0,C 180,E1 -13372.148,E2 -13372.148} C_VEL
LIN {X 0,Y 483.531,Z 939.234,A -85,B 0,C 180,E1 -13373.955,E2 -13373.955} C_VEL
LIN {X 0,Y 478.993,Z 957.794,A -85,B 0,C 180,E1 -13375.91,E2 -13375.91} C_VEL
LIN {X 0,Y 474.546,Z 975.305,A -85,B 0,C 180,E1 -13378.071,E2 -13378.071} C_VEL
LIN {X 0,Y 470.772,Z 990.397,A -85,B 0,C 180,E1 -13380.198,E2 -13380.198} C_VEL
LIN {X 0,Y 466.813,Z 1006.62,A -85,B 0,C 180,E1 -13382.855,E2 -13382.855} C_VEL
LIN {X 0,Y 463.859,Z 1019.408,A -85,B 0,C 180,E1 -13385.28,E2 -13385.28} C_VEL
LIN {X 0,Y 461.03,Z 1032.721,A -85,B 0,C 180,E1 -13388.231,E2 -13388.231} C_VEL
LIN {X 0,Y 459.196,Z 1042.603,A -85,B 0,C 180,E1 -13390.804,E2 -13390.804} C_VEL
LIN {X 0,Y 457.639,Z 1052.584,A -85,B 0,C 180,E1 -13393.89,E2 -13393.89} C_VEL
LIN {X 0,Y 456.771,Z 1059.687,A -85,B 0,C 180,E1 -13396.583,E2 -13396.583} C_VEL
LIN {X 0,Y 456.222,Z 1066.002,A -85,B 0,C 180,E1 -13399.519,E2 -13399.519} C_VEL
LIN {X 0,Y 455.988,Z 1070.568,A -85,B 0,C 180,E1 -13402.44,E2 -13402.44} C_VEL
LIN {X 0,Y 455.944,Z 1073.367,A -85,B 0,C 180,E1 -13404.967,E2 -13404.967} C_VEL
LIN {X 0,Y 455.937,Z 1075.275,A -85,B 0,C 180,E1 -13407.863,E2 -13407.863} C_VEL
LIN {X 0,Y 455.936,Z 1075.547,A -85,B 0,C 180,E1 -13410.754,E2 -13410.754} C_VEL
LIN {X 0,Y 455.94,Z 1074.65,A -85,B 0,C 180,E1 -13413.269,E2 -13413.269} C_VEL
LIN {X 0,Y 455.955,Z 1072.317,A -85,B 0,C 180,E1 -13416.169,E2 -13416.169} C_VEL
LIN {X 0,Y 456.077,Z 1068.334,A -85,B 0,C 180,E1 -13419.082,E2 -13419.082} C_VEL
LIN {X 0,Y 456.407,Z 1063.555,A -85,B 0,C 180,E1 -13421.682,E2 -13421.682} C_VEL
LIN {X 0,Y 457.138,Z 1056.522,A -85,B 0,C 180,E1 -13424.698,E2 -13424.698} C_VEL
LIN {X 0,Y 458.289,Z 1048.13,A -85,B 0,C 180,E1 -13427.551,E2 -13427.551} C_VEL
LIN {X 0,Y 460.063,Z 1037.89,A -85,B 0,C 180,E1 -13430.49,E2 -13430.49} C_VEL
LIN {X 0,Y 462.4,Z 1026.012,A -85,B 0,C 180,E1 -13433.311,E2 -13433.311} C_VEL
LIN {X 0,Y 465.346,Z 1012.949,A -85,B 0,C 180,E1 -13435.998,E2 -13435.998} C_VEL
LIN {X 0,Y 468.783,Z 998.36,A -85,B 0,C 180,E1 -13438.54,E2 -13438.54} C_VEL
LIN {X 0,Y 472.713,Z 982.664,A -85,B 0,C 180,E1 -13440.93,E2 -13440.93} C_VEL
LIN {X 0,Y 476.989,Z 965.468,A -85,B 0,C 180,E1 -13443.17,E2 -13443.17} C_VEL
LIN {X 0,Y 481.063,Z 949.208,A -85,B 0,C 180,E1 -13445.022,E2 -13445.022} C_VEL
LIN {X 0,Y 486.103,Z 928.478,A -85,B 0,C 180,E1 -13447.051,E2 -13447.051} C_VEL
LIN {X 0,Y 490.215,Z 910.75,A -85,B 0,C 180,E1 -13448.545,E2 -13448.545} C_VEL
LIN {X 0,Y 494.942,Z 888.977,A -85,B 0,C 180,E1 -13450.124,E2 -13450.124} C_VEL
LIN {X 0,Y 498.889,Z 869.138,A -85,B 0,C 180,E1 -13451.332,E2 -13451.332} C_VEL
LIN {X 0,Y 502.814,Z 847.448,A -85,B 0,C 180,E1 -13452.458,E2 -13452.458} C_VEL
LIN {X 0,Y 506.424,Z 823.984,A -85,B 0,C 180,E1 -13453.439,E2 -13453.439} C_VEL
LIN {X 0,Y 509.368,Z 801.882,A -85,B 0,C 180,E1 -13454.181,E2 -13454.181} C_VEL
LIN {X 0,Y 511.967,Z 776.657,A -85,B 0,C 180,E1 -13454.818,E2 -13454.818} C_VEL
LIN {X 0,Y 513.531,Z 754.139,A -85,B 0,C 180,E1 -13455.236,E2 -13455.236} C_VEL
LIN {X 0,Y 523.797,Z 504.981,A -85,B 0,C 180,E1 -13458.986,E2 -13458.986} C_VEL
LIN {X 0,Y 525.45,Z 464.206,A -85,B 0,C 180,E1 -13459.613,E2 -13459.613} C_VEL
LIN {X 0,Y 513.943,Z 444.342,A -85,B 0,C 180,E1 -13461.567,E2 -13461.567} C_VEL
LIN {X 0,Y 502.848,Z 426.624,A -85,B 0,C 180,E1 -13463.59,E2 -13463.59} C_VEL
LIN {X 0,Y 493.576,Z 412.822,A -85,B 0,C 180,E1 -13465.407,E2 -13465.407} C_VEL
LIN {X 0,Y 484.815,Z 400.364,A -85,B 0,C 180,E1 -13467.257,E2 -13467.257} C_VEL
LIN {X 0,Y 476.339,Z 388.949,A -85,B 0,C 180,E1 -13469.19,E2 -13469.19} C_VEL
LIN {X 0,Y 469.491,Z 380.088,A -85,B 0,C 180,E1 -13470.88,E2 -13470.88} C_VEL
LIN {X 0,Y 466.12,Z 375.516,A -85,B 0,C 180,E1 -13471.77,E2 -13471.77} C_VEL
LIN {X 0,Y 461.967,Z 370.709,A -85,B 0,C 180,E1 -13472.896,E2 -13472.896} C_VEL
LIN {X 0,Y 460.574,Z 368.866,A -85,B 0,C 180,E1 -13473.295,E2 -13473.295} C_VEL
LIN {X 0,Y 459.157,Z 367.071,A -85,B 0,C 180,E1 -13473.792,E2 -13473.792} C_VEL
LIN {X 0,Y 458.193,Z 364.144,A -85,B 0,C 180,E1 -13474.677,E2 -13474.677} C_VEL
LIN {X 0,Y 458.18,Z 364.155,A -85,B 0,C 180,E1 -13478.223,E2 -13478.223} C_VEL
LIN {X 0,Y 458.205,Z 364.158,A -85,B 0,C 180,E1 -13481.817,E2 -13481.817} C_VEL
LIN {X 0,Y 458.244,Z 364.142,A -85,B 0,C 180,E1 -13485.467,E2 -13485.467} C_VEL
LIN {X 0,Y 458.209,Z 364.132,A -85,B 0,C 180,E1 -13489.183,E2 -13489.183} C_VEL
LIN {X 0,Y 458.178,Z 364.126,A -85,B 0,C 180,E1 -13492.728,E2 -13492.728} C_VEL
LIN {X 0,Y 458.184,Z 364.136,A -85,B 0,C 180,E1 -13496.372,E2 -13496.372} C_VEL
LIN {X 0,Y 458.216,Z 364.153,A -85,B 0,C 180,E1 -13500,E2 -13500} C_VEL
LIN {X 0,Y 458.224,Z 364.141,A -85,B 0,C 180,E1 -13503.628,E2 -13503.628} C_VEL
LIN {X 0,Y 458.193,Z 364.126,A -85,B 0,C 180,E1 -13507.271,E2 -13507.271} C_VEL
LIN {X 0,Y 458.179,Z 364.13,A -85,B 0,C 180,E1 -13510.876,E2 -13510.876} C_VEL
LIN {X 0,Y 458.192,Z 364.143,A -85,B 0,C 180,E1 -13514.534,E2 -13514.534} C_VEL
LIN {X 0,Y 458.229,Z 364.152,A -85,B 0,C 180,E1 -13518.182,E2 -13518.182} C_VEL
LIN {X 0,Y 458.233,Z 364.151,A -85,B 0,C 180,E1 -13521.909,E2 -13521.909} C_VEL
LIN {X 0,Y 458.192,Z 364.147,A -85,B 0,C 180,E1 -13525.462,E2 -13525.462} C_VEL
LIN {X 0,Y 458.245,Z 364.318,A -85,B 0,C 180,E1 -13526.388,E2 -13526.388} C_VEL
LIN {X 0,Y 459.186,Z 367.116,A -85,B 0,C 180,E1 -13526.722,E2 -13526.722} C_VEL
LIN {X 0,Y 461.608,Z 369.749,A -85,B 0,C 180,E1 -13527.406,E2 -13527.406} C_VEL
LIN {X 0,Y 463.493,Z 370.954,A -85,B 0,C 180,E1 -13527.896,E2 -13527.896} C_VEL
LIN {X 0,Y 465.623,Z 374.584,A -85,B 0,C 180,E1 -13528.507,E2 -13528.507} C_VEL
LIN {X 0,Y 468.797,Z 377.436,A -85,B 0,C 180,E1 -13529.308,E2 -13529.308} C_VEL
LIN {X 0,Y 471.688,Z 381.458,A -85,B 0,C 180,E1 -13530.053,E2 -13530.053} C_VEL
LIN {X 0,Y 473.841,Z 383.618,A -85,B 0,C 180,E1 -13530.568,E2 -13530.568} C_VEL
LIN {X 0,Y 477.347,Z 387.978,A -85,B 0,C 180,E1 -13531.403,E2 -13531.403} C_VEL
LIN {X 0,Y 483.779,Z 396.033,A -85,B 0,C 180,E1 -13532.857,E2 -13532.857} C_VEL
LIN {X 0,Y 491.467,Z 405.768,A -85,B 0,C 180,E1 -13534.479,E2 -13534.479} C_VEL
LIN {X 0,Y 502.961,Z 421.168,A -85,B 0,C 180,E1 -13536.719,E2 -13536.719} C_VEL
LIN {X 0,Y 515.207,Z 438.813,A -85,B 0,C 180,E1 -13538.909,E2 -13538.909} C_VEL
LIN {X 0,Y 523.48,Z 451.997,A -85,B 0,C 180,E1 -13540.301,E2 -13540.301} C_VEL
LIN {X 0,Y 525.69,Z 456.214,A -85,B 0,C 180,E1 -13540.674,E2 -13540.674} C_VEL
LIN {X 0,Y 515.098,Z 709.677,A -85,B 0,C 180,E1 -13544.481,E2 -13544.481} C_VEL
LIN {X 0,Y 513.254,Z 748.312,A -85,B 0,C 180,E1 -13545.098,E2 -13545.098} C_VEL
LIN {X 0,Y 511.177,Z 771.845,A -85,B 0,C 180,E1 -13545.645,E2 -13545.645} C_VEL
LIN {X 0,Y 508.552,Z 795.306,A -85,B 0,C 180,E1 -13546.361,E2 -13546.361} C_VEL
LIN {X 0,Y 505.314,Z 817.927,A -85,B 0,C 180,E1 -13547.257,E2 -13547.257} C_VEL
LIN {X 0,Y 501.835,Z 839.243,A -85,B 0,C 180,E1 -13548.281,E2 -13548.281} C_VEL
LIN {X 0,Y 497.524,Z 861.933,A -85,B 0,C 180,E1 -13549.599,E2 -13549.599} C_VEL
LIN {X 0,Y 493.661,Z 880.504,A -85,B 0,C 180,E1 -13550.874,E2 -13550.874} C_VEL
LIN {X 0,Y 488.662,Z 902.573,A -85,B 0,C 180,E1 -13552.649,E2 -13552.649} C_VEL
LIN {X 0,Y 484.498,Z 919.735,A -85,B 0,C 180,E1 -13554.265,E2 -13554.265} C_VEL
LIN {X 0,Y 479.931,Z 937.971,A -85,B 0,C 180,E1 -13556.231,E2 -13556.231} C_VEL
LIN {X 0,Y 475.651,Z 954.337,A -85,B 0,C 180,E1 -13558.296,E2 -13558.296} C_VEL
LIN {X 0,Y 471.648,Z 969.908,A -85,B 0,C 180,E1 -13560.539,E2 -13560.539} C_VEL
LIN {X 0,Y 467.795,Z 984.843,A -85,B 0,C 180,E1 -13563.055,E2 -13563.055} C_VEL
LIN {X 0,Y 464.754,Z 997.28,A -85,B 0,C 180,E1 -13565.466,E2 -13565.466} C_VEL
LIN {X 0,Y 461.784,Z 1010.162,A -85,B 0,C 180,E1 -13568.402,E2 -13568.402} C_VEL
LIN {X 0,Y 459.82,Z 1019.716,A -85,B 0,C 180,E1 -13570.963,E2 -13570.963} C_VEL
LIN {X 0,Y 459.61,Z 1020.875,A -85,B 0,C 180,E1 -13571.292,E2 -13571.292} C_VEL
LIN {X 0,Y 458.102,Z 1023.946,A -85,B 0,C 180,E1 -13572.162,E2 -13572.162} C_VEL
LIN {X 0,Y 450.697,Z 1031.472,A -85,B 0,C 180,E1 -13574.491,E2 -13574.491} C_VEL
LIN {X 0,Y 449.627,Z 1033.607,A -85,B 0,C 180,E1 -13575.285,E2 -13575.285} C_VEL
LIN {X 0,Y 448.722,Z 1040.173,A -85,B 0,C 180,E1 -13578.301,E2 -13578.301} C_VEL
LIN {X 0,Y 448.27,Z 1044.838,A -85,B 0,C 180,E1 -13581.017,E2 -13581.017} C_VEL
LIN {X 0,Y 448.028,Z 1048.735,A -85,B 0,C 180,E1 -13584.236,E2 -13584.236} C_VEL
LIN {X 0,Y 447.962,Z 1050.607,A -85,B 0,C 180,E1 -13586.801,E2 -13586.801} C_VEL
LIN {X 0,Y 447.939,Z 1051.439,A -85,B 0,C 180,E1 -13589.361,E2 -13589.361} C_VEL
LIN {X 0,Y 447.956,Z 1051.057,A -85,B 0,C 180,E1 -13592.431,E2 -13592.431} C_VEL
LIN {X 0,Y 448.005,Z 1049.263,A -85,B 0,C 180,E1 -13595.25,E2 -13595.25} C_VEL
LIN {X 0,Y 448.142,Z 1046.528,A -85,B 0,C 180,E1 -13597.84,E2 -13597.84} C_VEL
LIN {X 0,Y 448.583,Z 1041.603,A -85,B 0,C 180,E1 -13601.052,E2 -13601.052} C_VEL
LIN {X 0,Y 449.27,Z 1035.982,A -85,B 0,C 180,E1 -13603.777,E2 -13603.777} C_VEL
LIN {X 0,Y 450.498,Z 1028.396,A -85,B 0,C 180,E1 -13606.771,E2 -13606.771} C_VEL
LIN {X 0,Y 452.307,Z 1018.903,A -85,B 0,C 180,E1 -13609.769,E2 -13609.769} C_VEL
LIN {X 0,Y 454.701,Z 1008.202,A -85,B 0,C 180,E1 -13612.633,E2 -13612.633} C_VEL
LIN {X 0,Y 457.646,Z 996.06,A -85,B 0,C 180,E1 -13615.356,E2 -13615.356} C_VEL
LIN {X 0,Y 460.79,Z 983.984,A -85,B 0,C 180,E1 -13617.706,E2 -13617.706} C_VEL
LIN {X 0,Y 465.034,Z 968.204,A -85,B 0,C 180,E1 -13620.35,E2 -13620.35} C_VEL
LIN {X 0,Y 469.048,Z 953.358,A -85,B 0,C 180,E1 -13622.493,E2 -13622.493} C_VEL
LIN {X 0,Y 474.036,Z 934.935,A -85,B 0,C 180,E1 -13624.79,E2 -13624.79} C_VEL
LIN {X 0,Y 478.344,Z 918.367,A -85,B 0,C 180,E1 -13626.565,E2 -13626.565} C_VEL
LIN {X 0,Y 483.21,Z 899.034,A -85,B 0,C 180,E1 -13628.373,E2 -13628.373} C_VEL
LIN {X 0,Y 487.887,Z 878.674,A -85,B 0,C 180,E1 -13629.978,E2 -13629.978} C_VEL
LIN {X 0,Y 492.323,Z 857.973,A -85,B 0,C 180,E1 -13631.382,E2 -13631.382} C_VEL
LIN {X 0,Y 496.618,Z 835.327,A -85,B 0,C 180,E1 -13632.649,E2 -13632.649} C_VEL
LIN {X 0,Y 500.258,Z 813.441,A -85,B 0,C 180,E1 -13633.675,E2 -13633.675} C_VEL
LIN {X 0,Y 503.565,Z 789.417,A -85,B 0,C 180,E1 -13634.569,E2 -13634.569} C_VEL
LIN {X 0,Y 506.037,Z 767.377,A -85,B 0,C 180,E1 -13635.213,E2 -13635.213} C_VEL
LIN {X 0,Y 508.109,Z 741.619,A -85,B 0,C 180,E1 -13635.76,E2 -13635.76} C_VEL
LIN {X 0,Y 518.11,Z 511.527,A -85,B 0,C 180,E1 -13639.26,E2 -13639.26} C_VEL
LIN {X 0,Y 520.318,Z 459.227,A -85,B 0,C 180,E1 -13640.07,E2 -13640.07} C_VEL
LIN {X 0,Y 512.266,Z 446.138,A -85,B 0,C 180,E1 -13641.454,E2 -13641.454} C_VEL
LIN {X 0,Y 500.856,Z 429.372,A -85,B 0,C 180,E1 -13643.529,E2 -13643.529} C_VEL
LIN {X 0,Y 490.179,Z 414.927,A -85,B 0,C 180,E1 -13645.63,E2 -13645.63} C_VEL
LIN {X 0,Y 482.289,Z 404.689,A -85,B 0,C 180,E1 -13647.311,E2 -13647.311} C_VEL
LIN {X 0,Y 478.648,Z 400.077,A -85,B 0,C 180,E1 -13648.13,E2 -13648.13} C_VEL
LIN {X 0,Y 474.297,Z 394.645,A -85,B 0,C 180,E1 -13649.149,E2 -13649.149} C_VEL
LIN {X 0,Y 470.19,Z 389.521,A -85,B 0,C 180,E1 -13650.157,E2 -13650.157} C_VEL
LIN {X 0,Y 466.724,Z 385.404,A -85,B 0,C 180,E1 -13651.041,E2 -13651.041} C_VEL
LIN {X 0,Y 465.456,Z 383.826,A -85,B 0,C 180,E1 -13651.377,E2 -13651.377} C_VEL
LIN {X 0,Y 462.189,Z 380.369,A -85,B 0,C 180,E1 -13652.246,E2 -13652.246} C_VEL
LIN {X 0,Y 460.728,Z 377.959,A -85,B 0,C 180,E1 -13652.677,E2 -13652.677} C_VEL
LIN {X 0,Y 457.536,Z 375.288,A -85,B 0,C 180,E1 -13653.559,E2 -13653.559} C_VEL
LIN {X 0,Y 455.422,Z 371.655,A -85,B 0,C 180,E1 -13654.233,E2 -13654.233} C_VEL
LIN {X 0,Y 452.353,Z 369.623,A -85,B 0,C 180,E1 -13655.132,E2 -13655.132} C_VEL
LIN {X 0,Y 450.66,Z 366.751,A -85,B 0,C 180,E1 -13655.713,E2 -13655.713} C_VEL
LIN {X 0,Y 450.29,Z 365.116,A -85,B 0,C 180,E1 -13655.884,E2 -13655.884} C_VEL
LIN {X 0,Y 450.253,Z 365.124,A -85,B 0,C 180,E1 -13659.459,E2 -13659.459} C_VEL
LIN {X 0,Y 450.239,Z 365.137,A -85,B 0,C 180,E1 -13663.087,E2 -13663.087} C_VEL
LIN {X 0,Y 450.247,Z 365.147,A -85,B 0,C 180,E1 -13666.777,E2 -13666.777} C_VEL
LIN {X 0,Y 450.274,Z 365.124,A -85,B 0,C 180,E1 -13670.413,E2 -13670.413} C_VEL
LIN {X 0,Y 450.277,Z 365.111,A -85,B 0,C 180,E1 -13674.009,E2 -13674.009} C_VEL
LIN {X 0,Y 450.243,Z 365.121,A -85,B 0,C 180,E1 -13677.582,E2 -13677.582} C_VEL
LIN {X 0,Y 450.24,Z 365.143,A -85,B 0,C 180,E1 -13681.273,E2 -13681.273} C_VEL
LIN {X 0,Y 450.252,Z 365.14,A -85,B 0,C 180,E1 -13684.969,E2 -13684.969} C_VEL
LIN {X 0,Y 450.288,Z 365.115,A -85,B 0,C 180,E1 -13688.556,E2 -13688.556} C_VEL
LIN {X 0,Y 450.275,Z 365.112,A -85,B 0,C 180,E1 -13692.309,E2 -13692.309} C_VEL
LIN {X 0,Y 450.243,Z 365.121,A -85,B 0,C 180,E1 -13695.852,E2 -13695.852} C_VEL
LIN {X 0,Y 450.237,Z 365.128,A -85,B 0,C 180,E1 -13699.593,E2 -13699.593} C_VEL
LIN {X 0,Y 450.259,Z 365.133,A -85,B 0,C 180,E1 -13703.166,E2 -13703.166} C_VEL
LIN {X 0,Y 450.279,Z 365.4,A -85,B 0,C 180,E1 -13703.493,E2 -13703.493} C_VEL
LIN {X 0,Y 450.973,Z 367.598,A -85,B 0,C 180,E1 -13704.077,E2 -13704.077} C_VEL
LIN {X 0,Y 453.166,Z 370.324,A -85,B 0,C 180,E1 -13704.786,E2 -13704.786} C_VEL
LIN {X 0,Y 454.703,Z 371.809,A -85,B 0,C 180,E1 -13705.252,E2 -13705.252} C_VEL
LIN {X 0,Y 459.451,Z 377.665,A -85,B 0,C 180,E1 -13706.671,E2 -13706.671} C_VEL
LIN {X 0,Y 463.009,Z 381.867,A -85,B 0,C 180,E1 -13707.665,E2 -13707.665} C_VEL
LIN {X 0,Y 467.387,Z 387.592,A -85,B 0,C 180,E1 -13708.844,E2 -13708.844} C_VEL
LIN {X 0,Y 476.281,Z 399.505,A -85,B 0,C 180,E1 -13711.059,E2 -13711.059} C_VEL
LIN {X 0,Y 485.623,Z 412.395,A -85,B 0,C 180,E1 -13713.174,E2 -13713.174} C_VEL
LIN {X 0,Y 497.083,Z 429.358,A -85,B 0,C 180,E1 -13715.544,E2 -13715.544} C_VEL
LIN {X 0,Y 507.745,Z 446.302,A -85,B 0,C 180,E1 -13717.571,E2 -13717.571} C_VEL
LIN {X 0,Y 518.685,Z 465.059,A -85,B 0,C 180,E1 -13719.506,E2 -13719.506} C_VEL
LIN {X 0,Y 520.257,Z 468.335,A -85,B 0,C 180,E1 -13719.783,E2 -13719.783} C_VEL
LIN {X 0,Y 509.613,Z 715.466,A -85,B 0,C 180,E1 -13723.524,E2 -13723.524} C_VEL
LIN {X 0,Y 507.288,Z 765.913,A -85,B 0,C 180,E1 -13724.316,E2 -13724.316} C_VEL
LIN {X 0,Y 504.993,Z 790.319,A -85,B 0,C 180,E1 -13724.864,E2 -13724.864} C_VEL
LIN {X 0,Y 502.454,Z 811.329,A -85,B 0,C 180,E1 -13725.479,E2 -13725.479} C_VEL
LIN {X 0,Y 498.796,Z 835.865,A -85,B 0,C 180,E1 -13726.403,E2 -13726.403} C_VEL
LIN {X 0,Y 495.455,Z 855.281,A -85,B 0,C 180,E1 -13727.305,E2 -13727.305} C_VEL
LIN {X 0,Y 491.289,Z 877.019,A -85,B 0,C 180,E1 -13728.501,E2 -13728.501} C_VEL
LIN {X 0,Y 486.703,Z 898.116,A -85,B 0,C 180,E1 -13729.905,E2 -13729.905} C_VEL
LIN {X 0,Y 482.182,Z 917.749,A -85,B 0,C 180,E1 -13731.424,E2 -13731.424} C_VEL
LIN {X 0,Y 477.187,Z 937.856,A -85,B 0,C 180,E1 -13733.257,E2 -13733.257} C_VEL
LIN {X 0,Y 472.856,Z 954.778,A -85,B 0,C 180,E1 -13735.037,E2 -13735.037} C_VEL
LIN {X 0,Y 467.794,Z 974.152,A -85,B 0,C 180,E1 -13737.409,E2 -13737.409} C_VEL
LIN {X 0,Y 464.03,Z 988.47,A -85,B 0,C 180,E1 -13739.434,E2 -13739.434} C_VEL
LIN {X 0,Y 459.995,Z 1004.274,A -85,B 0,C 180,E1 -13741.997,E2 -13741.997} C_VEL
LIN {X 0,Y 456.791,Z 1017.26,A -85,B 0,C 180,E1 -13744.455,E2 -13744.455} C_VEL
LIN {X 0,Y 453.949,Z 1029.877,A -85,B 0,C 180,E1 -13747.191,E2 -13747.191} C_VEL
LIN {X 0,Y 451.665,Z 1040.986,A -85,B 0,C 180,E1 -13750.067,E2 -13750.067} C_VEL
LIN {X 0,Y 450.114,Z 1050.074,A -85,B 0,C 180,E1 -13752.815,E2 -13752.815} C_VEL
LIN {X 0,Y 448.943,Z 1058.544,A -85,B 0,C 180,E1 -13755.95,E2 -13755.95} C_VEL
LIN {X 0,Y 448.349,Z 1064.492,A -85,B 0,C 180,E1 -13758.682,E2 -13758.682} C_VEL
LIN {X 0,Y 448.014,Z 1069.864,A -85,B 0,C 180,E1 -13761.917,E2 -13761.917} C_VEL
LIN {X 0,Y 447.946,Z 1072.921,A -85,B 0,C 180,E1 -13764.62,E2 -13764.62} C_VEL
LIN {X 0,Y 447.94,Z 1074.716,A -85,B 0,C 180,E1 -13767.185,E2 -13767.185} C_VEL
LIN {X 0,Y 447.94,Z 1075.425,A -85,B 0,C 180,E1 -13770.256,E2 -13770.256} C_VEL
LIN {X 0,Y 447.942,Z 1074.575,A -85,B 0,C 180,E1 -13773.071,E2 -13773.071} C_VEL
LIN {X 0,Y 447.949,Z 1072.684,A -85,B 0,C 180,E1 -13775.636,E2 -13775.636} C_VEL
LIN {X 0,Y 448.056,Z 1068.96,A -85,B 0,C 180,E1 -13778.728,E2 -13778.728} C_VEL
LIN {X 0,Y 448.388,Z 1063.966,A -85,B 0,C 180,E1 -13781.578,E2 -13781.578} C_VEL
LIN {X 0,Y 449.043,Z 1057.725,A -85,B 0,C 180,E1 -13784.39,E2 -13784.39} C_VEL
LIN {X 0,Y 450.304,Z 1048.823,A -85,B 0,C 180,E1 -13787.577,E2 -13787.577} C_VEL
LIN {X 0,Y 451.881,Z 1039.848,A -85,B 0,C 180,E1 -13790.248,E2 -13790.248} C_VEL
LIN {X 0,Y 454.42,Z 1027.533,A -85,B 0,C 180,E1 -13793.332,E2 -13793.332} C_VEL
LIN {X 0,Y 457.097,Z 1015.944,A -85,B 0,C 180,E1 -13795.805,E2 -13795.805} C_VEL
LIN {X 0,Y 460.736,Z 1001.253,A -85,B 0,C 180,E1 -13798.518,E2 -13798.518} C_VEL
LIN {X 0,Y 464.471,Z 986.711,A -85,B 0,C 180,E1 -13800.821,E2 -13800.821} C_VEL
LIN {X 0,Y 468.927,Z 969.848,A -85,B 0,C 180,E1 -13803.157,E2 -13803.157} C_VEL
LIN {X 0,Y 473.558,Z 951.903,A -85,B 0,C 180,E1 -13805.273,E2 -13805.273} C_VEL
LIN {X 0,Y 478.488,Z 932.783,A -85,B 0,C 180,E1 -13807.234,E2 -13807.234} C_VEL
LIN {X 0,Y 483.305,Z 912.746,A -85,B 0,C 180,E1 -13808.971,E2 -13808.971} C_VEL
LIN {X 0,Y 487.803,Z 893.086,A -85,B 0,C 180,E1 -13810.448,E2 -13810.448} C_VEL
LIN {X 0,Y 492.389,Z 871.069,A -85,B 0,C 180,E1 -13811.834,E2 -13811.834} C_VEL
LIN {X 0,Y 496.104,Z 851.36,A -85,B 0,C 180,E1 -13812.884,E2 -13812.884} C_VEL
LIN {X 0,Y 500.064,Z 827.464,A -85,B 0,C 180,E1 -13813.934,E2 -13813.934} C_VEL
LIN {X 0,Y 503.088,Z 805.815,A -85,B 0,C 180,E1 -13814.689,E2 -13814.689} C_VEL
LIN {X 0,Y 505.829,Z 782.137,A -85,B 0,C 180,E1 -13815.336,E2 -13815.336} C_VEL
LIN {X 0,Y 507.686,Z 757.769,A -85,B 0,C 180,E1 -13815.814,E2 -13815.814} C_VEL
LIN {X 0,Y 517.925,Z 518.885,A -85,B 0,C 180,E1 -13819.443,E2 -13819.443} C_VEL
LIN {X 0,Y 520.107,Z 467.74,A -85,B 0,C 180,E1 -13820.23,E2 -13820.23} C_VEL
LIN {X 0,Y 508.778,Z 448.073,A -85,B 0,C 180,E1 -13822.217,E2 -13822.217} C_VEL
LIN {X 0,Y 498.495,Z 431.686,A -85,B 0,C 180,E1 -13824.147,E2 -13824.147} C_VEL
LIN {X 0,Y 489.986,Z 418.848,A -85,B 0,C 180,E1 -13825.862,E2 -13825.862} C_VEL
LIN {X 0,Y 481.463,Z 406.639,A -85,B 0,C 180,E1 -13827.707,E2 -13827.707} C_VEL
LIN {X 0,Y 473.45,Z 395.688,A -85,B 0,C 180,E1 -13829.58,E2 -13829.58} C_VEL
LIN {X 0,Y 466.801,Z 387,A -85,B 0,C 180,E1 -13831.257,E2 -13831.257} C_VEL
LIN {X 0,Y 462.638,Z 381.536,A -85,B 0,C 180,E1 -13832.381,E2 -13832.381} C_VEL
LIN {X 0,Y 459.199,Z 377.276,A -85,B 0,C 180,E1 -13833.349,E2 -13833.349} C_VEL
LIN {X 0,Y 453.768,Z 370.789,A -85,B 0,C 180,E1 -13834.971,E2 -13834.971} C_VEL
LIN {X 0,Y 451.236,Z 368.072,A -85,B 0,C 180,E1 -13835.764,E2 -13835.764} C_VEL
LIN {X 0,Y 450.547,Z 366.526,A -85,B 0,C 180,E1 -13836.112,E2 -13836.112} C_VEL
LIN {X 0,Y 450.245,Z 365.123,A -85,B 0,C 180,E1 -13836.577,E2 -13836.577} C_VEL
LIN {X 0,Y 450.239,Z 365.122,A -85,B 0,C 180,E1 -13840.325,E2 -13840.325} C_VEL
LIN {X 0,Y 450.258,Z 365.116,A -85,B 0,C 180,E1 -13843.884,E2 -13843.884} C_VEL
LIN {X 0,Y 450.289,Z 365.116,A -85,B 0,C 180,E1 -13847.431,E2 -13847.431} C_VEL
LIN {X 0,Y 450.27,Z 365.132,A -85,B 0,C 180,E1 -13851.186,E2 -13851.186} C_VEL
LIN {X 0,Y 450.245,Z 365.147,A -85,B 0,C 180,E1 -13854.776,E2 -13854.776} C_VEL
LIN {X 0,Y 450.241,Z 365.127,A -85,B 0,C 180,E1 -13858.6,E2 -13858.6} C_VEL
LIN {X 0,Y 450.261,Z 365.112,A -85,B 0,C 180,E1 -13862.164,E2 -13862.164} C_VEL
LIN {X 0,Y 450.292,Z 365.115,A -85,B 0,C 180,E1 -13865.863,E2 -13865.863} C_VEL
LIN {X 0,Y 450.268,Z 365.142,A -85,B 0,C 180,E1 -13869.458,E2 -13869.458} C_VEL
LIN {X 0,Y 450.246,Z 365.139,A -85,B 0,C 180,E1 -13873.092,E2 -13873.092} C_VEL
LIN {X 0,Y 450.246,Z 365.125,A -85,B 0,C 180,E1 -13876.834,E2 -13876.834} C_VEL
LIN {X 0,Y 450.271,Z 365.116,A -85,B 0,C 180,E1 -13880.429,E2 -13880.429} C_VEL
LIN {X 0,Y 450.289,Z 365.115,A -85,B 0,C 180,E1 -13883.977,E2 -13883.977} C_VEL
LIN {X 0,Y 450.311,Z 365.305,A -85,B 0,C 180,E1 -13884.291,E2 -13884.291} C_VEL
LIN {X 0,Y 451.317,Z 368.217,A -85,B 0,C 180,E1 -13884.685,E2 -13884.685} C_VEL
LIN {X 0,Y 453.761,Z 370.807,A -85,B 0,C 180,E1 -13885.448,E2 -13885.448} C_VEL
LIN {X 0,Y 455.723,Z 372.048,A -85,B 0,C 180,E1 -13886.011,E2 -13886.011} C_VEL
LIN {X 0,Y 457.807,Z 375.623,A -85,B 0,C 180,E1 -13886.669,E2 -13886.669} C_VEL
LIN {X 0,Y 461.112,Z 378.515,A -85,B 0,C 180,E1 -13887.578,E2 -13887.578} C_VEL
LIN {X 0,Y 463.831,Z 382.416,A -85,B 0,C 180,E1 -13888.346,E2 -13888.346} C_VEL
LIN {X 0,Y 466.319,Z 384.757,A -85,B 0,C 180,E1 -13888.986,E2 -13888.986} C_VEL
LIN {X 0,Y 469.642,Z 389.039,A -85,B 0,C 180,E1 -13889.846,E2 -13889.846} C_VEL
LIN {X 0,Y 471.312,Z 390.883,A -85,B 0,C 180,E1 -13890.256,E2 -13890.256} C_VEL
LIN {X 0,Y 476.262,Z 397.104,A -85,B 0,C 180,E1 -13891.448,E2 -13891.448} C_VEL
LIN {X 0,Y 481.153,Z 403.252,A -85,B 0,C 180,E1 -13892.563,E2 -13892.563} C_VEL
LIN {X 0,Y 488.522,Z 412.697,A -85,B 0,C 180,E1 -13894.148,E2 -13894.148} C_VEL
LIN {X 0,Y 499.646,Z 427.749,A -85,B 0,C 180,E1 -13896.36,E2 -13896.36} C_VEL
LIN {X 0,Y 511.703,Z 445.332,A -85,B 0,C 180,E1 -13898.561,E2 -13898.561} C_VEL
LIN {X 0,Y 519.963,Z 458.699,A -85,B 0,C 180,E1 -13899.981,E2 -13899.981} C_VEL
LIN {X 0,Y 520.353,Z 459.963,A -85,B 0,C 180,E1 -13900.059,E2 -13900.059} C_VEL
LIN {X 0,Y 509.321,Z 714.8,A -85,B 0,C 180,E1 -13903.913,E2 -13903.913} C_VEL
LIN {X 0,Y 507.519,Z 749.678,A -85,B 0,C 180,E1 -13904.485,E2 -13904.485} C_VEL
LIN {X 0,Y 505.438,Z 772.463,A -85,B 0,C 180,E1 -13905.02,E2 -13905.02} C_VEL
LIN {X 0,Y 502.666,Z 796.313,A -85,B 0,C 180,E1 -13905.757,E2 -13905.757} C_VEL
LIN {X 0,Y 499.432,Z 818.151,A -85,B 0,C 180,E1 -13906.63,E2 -13906.63} C_VEL
LIN {X 0,Y 495.841,Z 839.467,A -85,B 0,C 180,E1 -13907.66,E2 -13907.66} C_VEL
LIN {X 0,Y 491.385,Z 862.155,A -85,B 0,C 180,E1 -13908.987,E2 -13908.987} C_VEL
LIN {X 0,Y 487.28,Z 881.236,A -85,B 0,C 180,E1 -13910.309,E2 -13910.309} C_VEL
LIN {X 0,Y 482.048,Z 903.457,A -85,B 0,C 180,E1 -13912.122,E2 -13912.122} C_VEL
LIN {X 0,Y 477.744,Z 920.561,A -85,B 0,C 180,E1 -13913.754,E2 -13913.754} C_VEL
LIN {X 0,Y 472.78,Z 939.498,A -85,B 0,C 180,E1 -13915.84,E2 -13915.84} C_VEL
LIN {X 0,Y 468.443,Z 955.476,A -85,B 0,C 180,E1 -13917.894,E2 -13917.894} C_VEL
LIN {X 0,Y 464.081,Z 971.743,A -85,B 0,C 180,E1 -13920.294,E2 -13920.294} C_VEL
LIN {X 0,Y 460.297,Z 985.757,A -85,B 0,C 180,E1 -13922.719,E2 -13922.719} C_VEL
LIN {X 0,Y 456.991,Z 998.755,A -85,B 0,C 180,E1 -13925.298,E2 -13925.298} C_VEL
LIN {X 0,Y 454.041,Z 1010.89,A -85,B 0,C 180,E1 -13928.15,E2 -13928.15} C_VEL
LIN {X 0,Y 451.908,Z 1020.84,A -85,B 0,C 180,E1 -13930.885,E2 -13930.885} C_VEL
LIN {X 0,Y 450.154,Z 1030.225,A -85,B 0,C 180,E1 -13934.012,E2 -13934.012} C_VEL
LIN {X 0,Y 449.627,Z 1033.607,A -85,B 0,C 180,E1 -13935.285,E2 -13935.285} C_VEL
LIN {X 0,Y 448.307,Z 1035.976,A -85,B 0,C 180,E1 -13936.214,E2 -13936.214} C_VEL
LIN {X 0,Y 441.274,Z 1041.737,A -85,B 0,C 180,E1 -13938.773,E2 -13938.773} C_VEL
LIN {X 0,Y 440.492,Z 1043.04,A -85,B 0,C 180,E1 -13939.544,E2 -13939.544} C_VEL
LIN {X 0,Y 440.146,Z 1047.118,A -85,B 0,C 180,E1 -13942.429,E2 -13942.429} C_VEL
LIN {X 0,Y 440.002,Z 1049.84,A -85,B 0,C 180,E1 -13945.177,E2 -13945.177} C_VEL
LIN {X 0,Y 439.945,Z 1051.475,A -85,B 0,C 180,E1 -13948.307,E2 -13948.307} C_VEL
LIN {X 0,Y 439.953,Z 1051.601,A -85,B 0,C 180,E1 -13951.042,E2 -13951.042} C_VEL
LIN {X 0,Y 439.973,Z 1050.671,A -85,B 0,C 180,E1 -13953.648,E2 -13953.648} C_VEL
LIN {X 0,Y 440.084,Z 1048.11,A -85,B 0,C 180,E1 -13956.837,E2 -13956.837} C_VEL
LIN {X 0,Y 440.362,Z 1044.391,A -85,B 0,C 180,E1 -13959.673,E2 -13959.673} C_VEL
LIN {X 0,Y 440.905,Z 1039.573,A -85,B 0,C 180,E1 -13962.442,E2 -13962.442} C_VEL
LIN {X 0,Y 442.034,Z 1032.084,A -85,B 0,C 180,E1 -13965.75,E2 -13965.75} C_VEL
LIN {X 0,Y 443.425,Z 1024.665,A -85,B 0,C 180,E1 -13968.403,E2 -13968.403} C_VEL
LIN {X 0,Y 445.666,Z 1014.508,A -85,B 0,C 180,E1 -13971.451,E2 -13971.451} C_VEL
LIN {X 0,Y 448.363,Z 1003.396,A -85,B 0,C 180,E1 -13974.226,E2 -13974.226} C_VEL
LIN {X 0,Y 451.802,Z 990.612,A -85,B 0,C 180,E1 -13976.981,E2 -13976.981} C_VEL
LIN {X 0,Y 455.717,Z 976.301,A -85,B 0,C 180,E1 -13979.582,E2 -13979.582} C_VEL
LIN {X 0,Y 460.273,Z 960.42,A -85,B 0,C 180,E1 -13982.088,E2 -13982.088} C_VEL
LIN {X 0,Y 464.91,Z 943.75,A -85,B 0,C 180,E1 -13984.322,E2 -13984.322} C_VEL
LIN {X 0,Y 469.915,Z 925.793,A -85,B 0,C 180,E1 -13986.417,E2 -13986.417} C_VEL
LIN {X 0,Y 474.779,Z 907.225,A -85,B 0,C 180,E1 -13988.255,E2 -13988.255} C_VEL
LIN {X 0,Y 479.336,Z 889.03,A -85,B 0,C 180,E1 -13989.822,E2 -13989.822} C_VEL
LIN {X 0,Y 484.352,Z 867.138,A -85,B 0,C 180,E1 -13991.425,E2 -13991.425} C_VEL
LIN {X 0,Y 488.083,Z 849.295,A -85,B 0,C 180,E1 -13992.535,E2 -13992.535} C_VEL
LIN {X 0,Y 492.331,Z 826.887,A -85,B 0,C 180,E1 -13993.723,E2 -13993.723} C_VEL
LIN {X 0,Y 495.873,Z 804.349,A -85,B 0,C 180,E1 -13994.687,E2 -13994.687} C_VEL
LIN {X 0,Y 498.729,Z 783.182,A -85,B 0,C 180,E1 -13995.422,E2 -13995.422} C_VEL
LIN {X 0,Y 501.329,Z 758.112,A -85,B 0,C 180,E1 -13996.086,E2 -13996.086} C_VEL
LIN {X 0,Y 502.875,Z 736.464,A -85,B 0,C 180,E1 -13996.505,E2 -13996.505} C_VEL
LIN {X 0,Y 514.141,Z 485.582,A -85,B 0,C 180,E1 -14000.334,E2 -14000.334} C_VEL
LIN {X 0,Y 515.064,Z 462.886,A -85,B 0,C 180,E1 -14000.699,E2 -14000.699} C_VEL
LIN {X 0,Y 507.046,Z 449.932,A -85,B 0,C 180,E1 -14002.118,E2 -14002.118} C_VEL
LIN {X 0,Y 495.249,Z 432.695,A -85,B 0,C 180,E1 -14004.34,E2 -14004.34} C_VEL
LIN {X 0,Y 484.087,Z 417.536,A -85,B 0,C 180,E1 -14006.637,E2 -14006.637} C_VEL
LIN {X 0,Y 475.721,Z 406.835,A -85,B 0,C 180,E1 -14008.513,E2 -14008.513} C_VEL
LIN {X 0,Y 471.424,Z 401.431,A -85,B 0,C 180,E1 -14009.541,E2 -14009.541} C_VEL
LIN {X 0,Y 467.257,Z 396.27,A -85,B 0,C 180,E1 -14010.586,E2 -14010.586} C_VEL
LIN {X 0,Y 463.663,Z 391.636,A -85,B 0,C 180,E1 -14011.537,E2 -14011.537} C_VEL
LIN {X 0,Y 459.797,Z 387.542,A -85,B 0,C 180,E1 -14012.582,E2 -14012.582} C_VEL
LIN {X 0,Y 458.129,Z 385.144,A -85,B 0,C 180,E1 -14013.071,E2 -14013.071} C_VEL
LIN {X 0,Y 454.83,Z 381.92,A -85,B 0,C 180,E1 -14014.022,E2 -14014.022} C_VEL
LIN {X 0,Y 453.094,Z 379.106,A -85,B 0,C 180,E1 -14014.582,E2 -14014.582} C_VEL
LIN {X 0,Y 449.921,Z 376.563,A -85,B 0,C 180,E1 -14015.549,E2 -14015.549} C_VEL
LIN {X 0,Y 447.979,Z 373.071,A -85,B 0,C 180,E1 -14016.242,E2 -14016.242} C_VEL
LIN {X 0,Y 444.191,Z 370.339,A -85,B 0,C 180,E1 -14017.5,E2 -14017.5} C_VEL
LIN {X 0,Y 442.606,Z 367.379,A -85,B 0,C 180,E1 -14018.132,E2 -14018.132} C_VEL
LIN {X 0,Y 442.333,Z 366.134,A -85,B 0,C 180,E1 -14018.289,E2 -14018.289} C_VEL
LIN {X 0,Y 442.35,Z 366.122,A -85,B 0,C 180,E1 -14021.96,E2 -14021.96} C_VEL
LIN {X 0,Y 442.316,Z 366.11,A -85,B 0,C 180,E1 -14025.601,E2 -14025.601} C_VEL
LIN {X 0,Y 442.298,Z 366.103,A -85,B 0,C 180,E1 -14029.185,E2 -14029.185} C_VEL
LIN {X 0,Y 442.303,Z 366.108,A -85,B 0,C 180,E1 -14032.943,E2 -14032.943} C_VEL
LIN {X 0,Y 442.326,Z 366.127,A -85,B 0,C 180,E1 -14036.631,E2 -14036.631} C_VEL
LIN {X 0,Y 442.358,Z 366.125,A -85,B 0,C 180,E1 -14040.389,E2 -14040.389} C_VEL
LIN {X 0,Y 442.341,Z 366.107,A -85,B 0,C 180,E1 -14044.278,E2 -14044.278} C_VEL
LIN {X 0,Y 442.311,Z 366.103,A -85,B 0,C 180,E1 -14047.926,E2 -14047.926} C_VEL
LIN {X 0,Y 442.298,Z 366.109,A -85,B 0,C 180,E1 -14051.607,E2 -14051.607} C_VEL
LIN {X 0,Y 442.302,Z 366.119,A -85,B 0,C 180,E1 -14055.337,E2 -14055.337} C_VEL
LIN {X 0,Y 442.327,Z 366.127,A -85,B 0,C 180,E1 -14058.997,E2 -14058.997} C_VEL
LIN {X 0,Y 442.325,Z 366.262,A -85,B 0,C 180,E1 -14061.355,E2 -14061.355} C_VEL
LIN {X 0,Y 443.491,Z 369.422,A -85,B 0,C 180,E1 -14061.909,E2 -14061.909} C_VEL
LIN {X 0,Y 446.078,Z 371.939,A -85,B 0,C 180,E1 -14062.817,E2 -14062.817} C_VEL
LIN {X 0,Y 447.718,Z 373.151,A -85,B 0,C 180,E1 -14063.354,E2 -14063.354} C_VEL
LIN {X 0,Y 450.706,Z 377.357,A -85,B 0,C 180,E1 -14064.371,E2 -14064.371} C_VEL
LIN {X 0,Y 452.687,Z 379.372,A -85,B 0,C 180,E1 -14064.988,E2 -14064.988} C_VEL
LIN {X 0,Y 457.186,Z 384.995,A -85,B 0,C 180,E1 -14066.358,E2 -14066.358} C_VEL
LIN {X 0,Y 461.5,Z 390.379,A -85,B 0,C 180,E1 -14067.588,E2 -14067.588} C_VEL
LIN {X 0,Y 468.982,Z 400.174,A -85,B 0,C 180,E1 -14069.576,E2 -14069.576} C_VEL
LIN {X 0,Y 476.777,Z 410.927,A -85,B 0,C 180,E1 -14071.48,E2 -14071.48} C_VEL
LIN {X 0,Y 485.588,Z 423.497,A -85,B 0,C 180,E1 -14073.459,E2 -14073.459} C_VEL
LIN {X 0,Y 494.678,Z 437.387,A -85,B 0,C 180,E1 -14075.352,E2 -14075.352} C_VEL
LIN {X 0,Y 504.353,Z 452.953,A -85,B 0,C 180,E1 -14077.223,E2 -14077.223} C_VEL
LIN {X 0,Y 514.91,Z 471.333,A -85,B 0,C 180,E1 -14079.132,E2 -14079.132} C_VEL
LIN {X 0,Y 505.212,Z 689.818,A -85,B 0,C 180,E1 -14082.475,E2 -14082.475} C_VEL
LIN {X 0,Y 501.862,Z 763.148,A -85,B 0,C 180,E1 -14083.616,E2 -14083.616} C_VEL
LIN {X 0,Y 499.535,Z 788.524,A -85,B 0,C 180,E1 -14084.169,E2 -14084.169} C_VEL
LIN {X 0,Y 497.033,Z 808.841,A -85,B 0,C 180,E1 -14084.754,E2 -14084.754} C_VEL
LIN {X 0,Y 493.421,Z 833.079,A -85,B 0,C 180,E1 -14085.643,E2 -14085.643} C_VEL
LIN {X 0,Y 489.939,Z 852.801,A -85,B 0,C 180,E1 -14086.546,E2 -14086.546} C_VEL
LIN {X 0,Y 486.015,Z 872.838,A -85,B 0,C 180,E1 -14087.633,E2 -14087.633} C_VEL
LIN {X 0,Y 481.053,Z 895.454,A -85,B 0,C 180,E1 -14089.1,E2 -14089.1} C_VEL
LIN {X 0,Y 476.798,Z 913.393,A -85,B 0,C 180,E1 -14090.471,E2 -14090.471} C_VEL
LIN {X 0,Y 471.777,Z 933.413,A -85,B 0,C 180,E1 -14092.236,E2 -14092.236} C_VEL
LIN {X 0,Y 466.809,Z 951.958,A -85,B 0,C 180,E1 -14094.165,E2 -14094.165} C_VEL
LIN {X 0,Y 461.893,Z 970.19,A -85,B 0,C 180,E1 -14096.346,E2 -14096.346} C_VEL
LIN {X 0,Y 457.38,Z 986.544,A -85,B 0,C 180,E1 -14098.648,E2 -14098.648} C_VEL
LIN {X 0,Y 453.47,Z 1001.077,A -85,B 0,C 180,E1 -14100.981,E2 -14100.981} C_VEL
LIN {X 0,Y 449.645,Z 1015.754,A -85,B 0,C 180,E1 -14103.735,E2 -14103.735} C_VEL
LIN {X 0,Y 446.83,Z 1027.336,A -85,B 0,C 180,E1 -14106.247,E2 -14106.247} C_VEL
LIN {X 0,Y 444.106,Z 1039.835,A -85,B 0,C 180,E1 -14109.437,E2 -14109.437} C_VEL
LIN {X 0,Y 442.468,Z 1048.621,A -85,B 0,C 180,E1 -14112.101,E2 -14112.101} C_VEL
LIN {X 0,Y 441.141,Z 1057.401,A -85,B 0,C 180,E1 -14115.294,E2 -14115.294} C_VEL
LIN {X 0,Y 440.449,Z 1063.507,A -85,B 0,C 180,E1 -14118.082,E2 -14118.082} C_VEL
LIN {X 0,Y 440.072,Z 1068.541,A -85,B 0,C 180,E1 -14120.98,E2 -14120.98} C_VEL
LIN {X 0,Y 439.953,Z 1072.358,A -85,B 0,C 180,E1 -14124.13,E2 -14124.13} C_VEL
LIN {X 0,Y 439.943,Z 1074.294,A -85,B 0,C 180,E1 -14126.743,E2 -14126.743} C_VEL
LIN {X 0,Y 439.941,Z 1075.167,A -85,B 0,C 180,E1 -14129.479,E2 -14129.479} C_VEL
LIN {X 0,Y 439.941,Z 1074.639,A -85,B 0,C 180,E1 -14132.605,E2 -14132.605} C_VEL
LIN {X 0,Y 439.947,Z 1072.818,A -85,B 0,C 180,E1 -14135.347,E2 -14135.347} C_VEL
LIN {X 0,Y 440.005,Z 1069.969,A -85,B 0,C 180,E1 -14137.968,E2 -14137.968} C_VEL
LIN {X 0,Y 440.34,Z 1064.785,A -85,B 0,C 180,E1 -14141.261,E2 -14141.261} C_VEL
LIN {X 0,Y 440.939,Z 1058.931,A -85,B 0,C 180,E1 -14144.042,E2 -14144.042} C_VEL
LIN {X 0,Y 442.075,Z 1051.051,A -85,B 0,C 180,E1 -14147.1,E2 -14147.1} C_VEL
LIN {X 0,Y 443.818,Z 1041.214,A -85,B 0,C 180,E1 -14150.163,E2 -14150.163} C_VEL
LIN {X 0,Y 446.072,Z 1030.695,A -85,B 0,C 180,E1 -14152.956,E2 -14152.956} C_VEL
LIN {X 0,Y 449.158,Z 1017.651,A -85,B 0,C 180,E1 -14155.869,E2 -14155.869} C_VEL
LIN {X 0,Y 452.482,Z 1004.721,A -85,B 0,C 180,E1 -14158.366,E2 -14158.366} C_VEL
LIN {X 0,Y 456.676,Z 989.05,A -85,B 0,C 180,E1 -14160.966,E2 -14160.966} C_VEL
LIN {X 0,Y 460.737,Z 974.197,A -85,B 0,C 180,E1 -14163.102,E2 -14163.102} C_VEL
LIN {X 0,Y 465.81,Z 955.598,A -85,B 0,C 180,E1 -14165.42,E2 -14165.42} C_VEL
LIN {X 0,Y 470.44,Z 938.154,A -85,B 0,C 180,E1 -14167.283,E2 -14167.283} C_VEL
LIN {X 0,Y 475.699,Z 917.774,A -85,B 0,C 180,E1 -14169.163,E2 -14169.163} C_VEL
LIN {X 0,Y 480.274,Z 898.575,A -85,B 0,C 180,E1 -14170.665,E2 -14170.665} C_VEL
LIN {X 0,Y 484.763,Z 878.578,A -85,B 0,C 180,E1 -14172.015,E2 -14172.015} C_VEL
LIN {X 0,Y 489.291,Z 856.004,A -85,B 0,C 180,E1 -14173.283,E2 -14173.283} C_VEL
LIN {X 0,Y 492.726,Z 836.706,A -85,B 0,C 180,E1 -14174.192,E2 -14174.192} C_VEL
LIN {X 0,Y 496.462,Z 812.753,A -85,B 0,C 180,E1 -14175.113,E2 -14175.113} C_VEL
LIN {X 0,Y 499.196,Z 790.891,A -85,B 0,C 180,E1 -14175.762,E2 -14175.762} C_VEL
LIN {X 0,Y 501.512,Z 767.25,A -85,B 0,C 180,E1 -14176.301,E2 -14176.301} C_VEL
LIN {X 0,Y 503.497,Z 728.024,A -85,B 0,C 180,E1 -14176.935,E2 -14176.935} C_VEL
LIN {X 0,Y 514.476,Z 480.818,A -85,B 0,C 180,E1 -14180.702,E2 -14180.702} C_VEL
LIN {X 0,Y 514.757,Z 471.16,A -85,B 0,C 180,E1 -14180.872,E2 -14180.872} C_VEL
LIN {X 0,Y 504.126,Z 452.66,A -85,B 0,C 180,E1 -14182.793,E2 -14182.793} C_VEL
LIN {X 0,Y 492.338,Z 433.611,A -85,B 0,C 180,E1 -14185.096,E2 -14185.096} C_VEL
LIN {X 0,Y 479.696,Z 414.867,A -85,B 0,C 180,E1 -14187.813,E2 -14187.813} C_VEL
LIN {X 0,Y 470.361,Z 402.144,A -85,B 0,C 180,E1 -14190.029,E2 -14190.029} C_VEL
LIN {X 0,Y 464.238,Z 394.024,A -85,B 0,C 180,E1 -14191.611,E2 -14191.611} C_VEL
LIN {X 0,Y 459.921,Z 388.389,A -85,B 0,C 180,E1 -14192.8,E2 -14192.8} C_VEL
LIN {X 0,Y 454.602,Z 381.726,A -85,B 0,C 180,E1 -14194.358,E2 -14194.358} C_VEL
LIN {X 0,Y 451.477,Z 378.041,A -85,B 0,C 180,E1 -14195.325,E2 -14195.325} C_VEL
LIN {X 0,Y 448.738,Z 374.798,A -85,B 0,C 180,E1 -14196.215,E2 -14196.215} C_VEL
LIN {X 0,Y 446.996,Z 372.428,A -85,B 0,C 180,E1 -14196.815,E2 -14196.815} C_VEL
LIN {X 0,Y 443.874,Z 369.969,A -85,B 0,C 180,E1 -14197.867,E2 -14197.867} C_VEL
LIN {X 0,Y 442.496,Z 367.14,A -85,B 0,C 180,E1 -14198.426,E2 -14198.426} C_VEL
LIN {X 0,Y 442.307,Z 366.12,A -85,B 0,C 180,E1 -14198.625,E2 -14198.625} C_VEL
LIN {X 0,Y 442.303,Z 366.127,A -85,B 0,C 180,E1 -14202.366,E2 -14202.366} C_VEL
LIN {X 0,Y 442.311,Z 366.136,A -85,B 0,C 180,E1 -14206.136,E2 -14206.136} C_VEL
LIN {X 0,Y 442.342,Z 366.117,A -85,B 0,C 180,E1 -14209.713,E2 -14209.713} C_VEL
LIN {X 0,Y 442.357,Z 366.1,A -85,B 0,C 180,E1 -14213.511,E2 -14213.511} C_VEL
LIN {X 0,Y 442.325,Z 366.1,A -85,B 0,C 180,E1 -14217.279,E2 -14217.279} C_VEL
LIN {X 0,Y 442.304,Z 366.118,A -85,B 0,C 180,E1 -14220.777,E2 -14220.777} C_VEL
LIN {X 0,Y 442.309,Z 366.136,A -85,B 0,C 180,E1 -14224.538,E2 -14224.538} C_VEL
LIN {X 0,Y 442.333,Z 366.114,A -85,B 0,C 180,E1 -14228.187,E2 -14228.187} C_VEL
LIN {X 0,Y 442.348,Z 366.099,A -85,B 0,C 180,E1 -14231.87,E2 -14231.87} C_VEL
LIN {X 0,Y 442.319,Z 366.105,A -85,B 0,C 180,E1 -14235.471,E2 -14235.471} C_VEL
LIN {X 0,Y 442.308,Z 366.114,A -85,B 0,C 180,E1 -14239.135,E2 -14239.135} C_VEL
LIN {X 0,Y 442.384,Z 366.335,A -85,B 0,C 180,E1 -14241.923,E2 -14241.923} C_VEL
LIN {X 0,Y 443.389,Z 369.2,A -85,B 0,C 180,E1 -14242.368,E2 -14242.368} C_VEL
LIN {X 0,Y 445.695,Z 371.708,A -85,B 0,C 180,E1 -14243.187,E2 -14243.187} C_VEL
LIN {X 0,Y 447.967,Z 373.075,A -85,B 0,C 180,E1 -14243.916,E2 -14243.916} C_VEL
LIN {X 0,Y 449.966,Z 376.619,A -85,B 0,C 180,E1 -14244.624,E2 -14244.624} C_VEL
LIN {X 0,Y 453.434,Z 379.55,A -85,B 0,C 180,E1 -14245.678,E2 -14245.678} C_VEL
LIN {X 0,Y 456.062,Z 383.424,A -85,B 0,C 180,E1 -14246.498,E2 -14246.498} C_VEL
LIN {X 0,Y 458.717,Z 385.81,A -85,B 0,C 180,E1 -14247.242,E2 -14247.242} C_VEL
LIN {X 0,Y 461.943,Z 390.094,A -85,B 0,C 180,E1 -14248.156,E2 -14248.156} C_VEL
LIN {X 0,Y 463.964,Z 392.173,A -85,B 0,C 180,E1 -14248.689,E2 -14248.689} C_VEL
LIN {X 0,Y 467.715,Z 396.712,A -85,B 0,C 180,E1 -14249.664,E2 -14249.664} C_VEL
LIN {X 0,Y 473.698,Z 404.315,A -85,B 0,C 180,E1 -14251.141,E2 -14251.141} C_VEL
LIN {X 0,Y 481.389,Z 413.985,A -85,B 0,C 180,E1 -14252.899,E2 -14252.899} C_VEL
LIN {X 0,Y 492.409,Z 428.857,A -85,B 0,C 180,E1 -14255.219,E2 -14255.219} C_VEL
LIN {X 0,Y 504.098,Z 445.546,A -85,B 0,C 180,E1 -14257.46,E2 -14257.46} C_VEL
LIN {X 0,Y 512.998,Z 459.502,A -85,B 0,C 180,E1 -14259.054,E2 -14259.054} C_VEL
LIN {X 0,Y 515.089,Z 463.377,A -85,B 0,C 180,E1 -14259.426,E2 -14259.426} C_VEL
LIN {X 0,Y 503.663,Z 718.343,A -85,B 0,C 180,E1 -14263.308,E2 -14263.308} C_VEL
LIN {X 0,Y 501.819,Z 751.356,A -85,B 0,C 180,E1 -14263.864,E2 -14263.864} C_VEL
LIN {X 0,Y 499.72,Z 773.471,A -85,B 0,C 180,E1 -14264.392,E2 -14264.392} C_VEL
LIN {X 0,Y 496.726,Z 798.011,A -85,B 0,C 180,E1 -14265.167,E2 -14265.167} C_VEL
LIN {X 0,Y 493.404,Z 819.654,A -85,B 0,C 180,E1 -14266.046,E2 -14266.046} C_VEL
LIN {X 0,Y 489.516,Z 841.939,A -85,B 0,C 180,E1 -14267.142,E2 -14267.142} C_VEL
LIN {X 0,Y 485.114,Z 863.272,A -85,B 0,C 180,E1 -14268.418,E2 -14268.418} C_VEL
LIN {X 0,Y 480.797,Z 882.645,A -85,B 0,C 180,E1 -14269.78,E2 -14269.78} C_VEL
LIN {X 0,Y 475.647,Z 903.68,A -85,B 0,C 180,E1 -14271.52,E2 -14271.52} C_VEL
LIN {X 0,Y 471.204,Z 920.723,A -85,B 0,C 180,E1 -14273.161,E2 -14273.161} C_VEL
LIN {X 0,Y 466.1,Z 939.499,A -85,B 0,C 180,E1 -14275.248,E2 -14275.248} C_VEL
LIN {X 0,Y 461.514,Z 955.698,A -85,B 0,C 180,E1 -14277.353,E2 -14277.353} C_VEL
LIN {X 0,Y 456.908,Z 972.156,A -85,B 0,C 180,E1 -14279.816,E2 -14279.816} C_VEL
LIN {X 0,Y 452.955,Z 986.16,A -85,B 0,C 180,E1 -14282.277,E2 -14282.277} C_VEL
LIN {X 0,Y 449.382,Z 999.6,A -85,B 0,C 180,E1 -14284.991,E2 -14284.991} C_VEL
LIN {X 0,Y 446.307,Z 1011.619,A -85,B 0,C 180,E1 -14287.89,E2 -14287.89} C_VEL
LIN {X 0,Y 443.998,Z 1021.964,A -85,B 0,C 180,E1 -14290.805,E2 -14290.805} C_VEL
LIN {X 0,Y 442.252,Z 1030.792,A -85,B 0,C 180,E1 -14293.854,E2 -14293.854} C_VEL
LIN {X 0,Y 441.187,Z 1037.471,A -85,B 0,C 180,E1 -14296.634,E2 -14296.634} C_VEL
LIN {X 0,Y 440.492,Z 1043.04,A -85,B 0,C 180,E1 -14299.544,E2 -14299.544} C_VEL
LIN {X 0,Y 439.356,Z 1044.611,A -85,B 0,C 180,E1 -14300.524,E2 -14300.524} C_VEL
LIN {X 0,Y 434.544,Z 1047.37,A -85,B 0,C 180,E1 -14302.369,E2 -14302.369} C_VEL
LIN {X 0,Y 432.222,Z 1048.856,A -85,B 0,C 180,E1 -14303.65,E2 -14303.65} C_VEL
LIN {X 0,Y 432.054,Z 1049.16,A -85,B 0,C 180,E1 -14304.016,E2 -14304.016} C_VEL
LIN {X 0,Y 431.972,Z 1051.035,A -85,B 0,C 180,E1 -14306.683,E2 -14306.683} C_VEL
LIN {X 0,Y 431.946,Z 1051.866,A -85,B 0,C 180,E1 -14309.337,E2 -14309.337} C_VEL
LIN {X 0,Y 431.961,Z 1051.484,A -85,B 0,C 180,E1 -14312.521,E2 -14312.521} C_VEL
LIN {X 0,Y 432.02,Z 1049.691,A -85,B 0,C 180,E1 -14315.445,E2 -14315.445} C_VEL
LIN {X 0,Y 432.182,Z 1046.978,A -85,B 0,C 180,E1 -14318.113,E2 -14318.113} C_VEL
LIN {X 0,Y 432.696,Z 1042.033,A -85,B 0,C 180,E1 -14321.463,E2 -14321.463} C_VEL
LIN {X 0,Y 433.505,Z 1036.253,A -85,B 0,C 180,E1 -14324.362,E2 -14324.362} C_VEL
LIN {X 0,Y 434.941,Z 1028.468,A -85,B 0,C 180,E1 -14327.527,E2 -14327.527} C_VEL
LIN {X 0,Y 436.903,Z 1019.337,A -85,B 0,C 180,E1 -14330.497,E2 -14330.497} C_VEL
LIN {X 0,Y 439.441,Z 1009.144,A -85,B 0,C 180,E1 -14333.323,E2 -14333.323} C_VEL
LIN {X 0,Y 442.839,Z 996.495,A -85,B 0,C 180,E1 -14336.267,E2 -14336.267} C_VEL
LIN {X 0,Y 446.448,Z 983.907,A -85,B 0,C 180,E1 -14338.785,E2 -14338.785} C_VEL
LIN {X 0,Y 451.167,Z 967.8,A -85,B 0,C 180,E1 -14341.536,E2 -14341.536} C_VEL
LIN {X 0,Y 455.588,Z 952.871,A -85,B 0,C 180,E1 -14343.729,E2 -14343.729} C_VEL
LIN {X 0,Y 461.036,Z 934.104,A -85,B 0,C 180,E1 -14346.096,E2 -14346.096} C_VEL
LIN {X 0,Y 465.657,Z 917.588,A -85,B 0,C 180,E1 -14347.888,E2 -14347.888} C_VEL
LIN {X 0,Y 471.115,Z 897.151,A -85,B 0,C 180,E1 -14349.798,E2 -14349.798} C_VEL
LIN {X 0,Y 475.759,Z 878.288,A -85,B 0,C 180,E1 -14351.294,E2 -14351.294} C_VEL
